LIN {X 0,Y 392.678,Z 1253.285,A -85,B 0,C 180,E1 10734.702,E2 10734.702} C_VEL
LIN {X 0,Y 397.853,Z 1224.84,A -85,B 0,C 180,E1 10739.855,E2 10739.855} C_VEL
LIN {X 0,Y 404.262,Z 1192.64,A -85,B 0,C 180,E1 10744.206,E2 10744.206} C_VEL
LIN {X 0,Y 411.173,Z 1158.01,A -85,B 0,C 180,E1 10747.665,E2 10747.665} C_VEL
LIN {X 0,Y 417.671,Z 1121.351,A -85,B 0,C 180,E1 10750.31,E2 10750.31} C_VEL
LIN {X 0,Y 423.279,Z 1083.5,A -85,B 0,C 180,E1 10752.143,E2 10752.143} C_VEL
LIN {X 0,Y 425.073,Z 1063.403,A -85,B 0,C 180,E1 10752.868,E2 10752.868} C_VEL
LIN {X 0,Y 408.001,Z 1028.181,A -85,B 0,C 180,E1 10756.188,E2 10756.188} C_VEL
LIN {X 0,Y 387.571,Z 994.661,A -85,B 0,C 180,E1 10760.209,E2 10760.209} C_VEL
LIN {X 0,Y 385.179,Z 989.03,A -85,B 0,C 180,E1 10760.945,E2 10760.945} C_VEL
LIN {X 0,Y 385.144,Z 989.03,A -85,B 0,C 180,E1 10766.736,E2 10766.736} C_VEL
LIN {X 0,Y 385.369,Z 989.03,A -85,B 0,C 180,E1 10774.238,E2 10774.238} C_VEL
LIN {X 0,Y 385.666,Z 989.03,A -85,B 0,C 180,E1 10779.892,E2 10779.892} C_VEL
LIN {X 0,Y 385.82,Z 989.03,A -85,B 0,C 180,E1 10786.428,E2 10786.428} C_VEL
LIN {X 0,Y 386.249,Z 989.03,A -85,B 0,C 180,E1 10793.269,E2 10793.269} C_VEL
LIN {X 0,Y 386.525,Z 989.03,A -85,B 0,C 180,E1 10800,E2 10800} C_VEL
LIN {X 0,Y 386.241,Z 989.03,A -85,B 0,C 180,E1 10806.731,E2 10806.731} C_VEL
LIN {X 0,Y 385.972,Z 989.03,A -85,B 0,C 180,E1 10813.566,E2 10813.566} C_VEL
LIN {X 0,Y 385.612,Z 989.03,A -85,B 0,C 180,E1 10820.621,E2 10820.621} C_VEL
LIN {X 0,Y 385.312,Z 989.03,A -85,B 0,C 180,E1 10828.03,E2 10828.03} C_VEL
LIN {X 0,Y 385.061,Z 989.03,A -85,B 0,C 180,E1 10834.619,E2 10834.619} C_VEL
LIN {X 0,Y 385.053,Z 989.03,A -85,B 0,C 180,E1 10838.83,E2 10838.83} C_VEL
LIN {X 0,Y 385.09,Z 989.144,A -85,B 0,C 180,E1 10842.934,E2 10842.934} C_VEL
LIN {X 0,Y 392.046,Z 1004.005,A -85,B 0,C 180,E1 10845.356,E2 10845.356} C_VEL
LIN {X 0,Y 402.939,Z 1029.34,A -85,B 0,C 180,E1 10849.545,E2 10849.545} C_VEL
LIN {X 0,Y 410.17,Z 1055.044,A -85,B 0,C 180,E1 10853.66,E2 10853.66} C_VEL
LIN {X 0,Y 411.018,Z 1064.8,A -85,B 0,C 180,E1 10855.123,E2 10855.123} C_VEL
LIN {X 0,Y 404.003,Z 1094.796,A -85,B 0,C 180,E1 10859.209,E2 10859.209} C_VEL
LIN {X 0,Y 397.397,Z 1120.838,A -85,B 0,C 180,E1 10864.108,E2 10864.108} C_VEL
LIN {X 0,Y 392.663,Z 1140.325,A -85,B 0,C 180,E1 10869.178,E2 10869.178} C_VEL
LIN {X 0,Y 389.485,Z 1155.427,A -85,B 0,C 180,E1 10874.758,E2 10874.758} C_VEL
LIN {X 0,Y 388.053,Z 1164.693,A -85,B 0,C 180,E1 10879.923,E2 10879.923} C_VEL
LIN {X 0,Y 387.281,Z 1170.266,A -85,B 0,C 180,E1 10885.531,E2 10885.531} C_VEL
LIN {X 0,Y 387.373,Z 1171.602,A -85,B 0,C 180,E1 10890.001,E2 10890.001} C_VEL
LIN {X 0,Y 387.286,Z 1170.199,A -85,B 0,C 180,E1 10894.47,E2 10894.47} C_VEL
LIN {X 0,Y 388.016,Z 1164.559,A -85,B 0,C 180,E1 10900.08,E2 10900.08} C_VEL
LIN {X 0,Y 389.699,Z 1154.162,A -85,B 0,C 180,E1 10905.728,E2 10905.728} C_VEL
LIN {X 0,Y 393.119,Z 1138.154,A -85,B 0,C 180,E1 10911.388,E2 10911.388} C_VEL
LIN {X 0,Y 398.156,Z 1117.854,A -85,B 0,C 180,E1 10916.445,E2 10916.445} C_VEL
LIN {X 0,Y 404.626,Z 1091.985,A -85,B 0,C 180,E1 10921.132,E2 10921.132} C_VEL
LIN {X 0,Y 411.178,Z 1062.825,A -85,B 0,C 180,E1 10925.038,E2 10925.038} C_VEL
LIN {X 0,Y 407.077,Z 1042.475,A -85,B 0,C 180,E1 10928.252,E2 10928.252} C_VEL
LIN {X 0,Y 397.567,Z 1015.888,A -85,B 0,C 180,E1 10932.556,E2 10932.556} C_VEL
LIN {X 0,Y 385.142,Z 989.03,A -85,B 0,C 180,E1 10936.979,E2 10936.979} C_VEL
LIN {X 0,Y 385.177,Z 989.03,A -85,B 0,C 180,E1 10944.011,E2 10944.011} C_VEL
LIN {X 0,Y 385.338,Z 989.03,A -85,B 0,C 180,E1 10951.972,E2 10951.972} C_VEL
LIN {X 0,Y 385.624,Z 989.03,A -85,B 0,C 180,E1 10959.38,E2 10959.38} C_VEL
LIN {X 0,Y 385.831,Z 989.03,A -85,B 0,C 180,E1 10966.429,E2 10966.429} C_VEL
LIN {X 0,Y 386.309,Z 989.03,A -85,B 0,C 180,E1 10973.271,E2 10973.271} C_VEL
LIN {X 0,Y 386.585,Z 989.03,A -85,B 0,C 180,E1 10980,E2 10980} C_VEL
LIN {X 0,Y 386.252,Z 989.03,A -85,B 0,C 180,E1 10986.731,E2 10986.731} C_VEL
LIN {X 0,Y 385.983,Z 989.03,A -85,B 0,C 180,E1 10993.566,E2 10993.566} C_VEL
LIN {X 0,Y 385.608,Z 989.03,A -85,B 0,C 180,E1 11000.621,E2 11000.621} C_VEL
LIN {X 0,Y 385.384,Z 989.03,A -85,B 0,C 180,E1 11008.025,E2 11008.025} C_VEL
LIN {X 0,Y 385.21,Z 989.03,A -85,B 0,C 180,E1 11014.648,E2 11014.648} C_VEL
LIN {X 0,Y 385.194,Z 989.03,A -85,B 0,C 180,E1 11019.234,E2 11019.234} C_VEL
LIN {X 0,Y 387.509,Z 994.603,A -85,B 0,C 180,E1 11019.796,E2 11019.796} C_VEL
LIN {X 0,Y 408.246,Z 1028.761,A -85,B 0,C 180,E1 11023.871,E2 11023.871} C_VEL
LIN {X 0,Y 425.015,Z 1063.2,A -85,B 0,C 180,E1 11027.121,E2 11027.121} C_VEL
LIN {X 0,Y 420.317,Z 1104.533,A -85,B 0,C 180,E1 11028.776,E2 11028.776} C_VEL
LIN {X 0,Y 414.189,Z 1141.892,A -85,B 0,C 180,E1 11031.062,E2 11031.062} C_VEL
LIN {X 0,Y 407.588,Z 1176.514,A -85,B 0,C 180,E1 11034.053,E2 11034.053} C_VEL
LIN {X 0,Y 400.807,Z 1210.155,A -85,B 0,C 180,E1 11038.008,E2 11038.008} C_VEL
LIN {X 0,Y 395.066,Z 1240.02,A -85,B 0,C 180,E1 11042.718,E2 11042.718} C_VEL
LIN {X 0,Y 390.9,Z 1264.641,A -85,B 0,C 180,E1 11047.887,E2 11047.887} C_VEL
LIN {X 0,Y 388.53,Z 1283,A -85,B 0,C 180,E1 11053.064,E2 11053.064} C_VEL
LIN {X 0,Y 387.502,Z 1297.201,A -85,B 0,C 180,E1 11058.771,E2 11058.771} C_VEL
LIN {X 0,Y 387.197,Z 1304.359,A -85,B 0,C 180,E1 11063.366,E2 11063.366} C_VEL
LIN {X 0,Y 385.864,Z 1305.49,A -85,B 0,C 180,E1 11064.634,E2 11064.634} C_VEL
LIN {X 0,Y 379.328,Z 1306.601,A -85,B 0,C 180,E1 11068.462,E2 11068.462} C_VEL
LIN {X 0,Y 379.401,Z 1306.453,A -85,B 0,C 180,E1 11072.279,E2 11072.279} C_VEL
LIN {X 0,Y 379.39,Z 1301.51,A -85,B 0,C 180,E1 11078.001,E2 11078.001} C_VEL
LIN {X 0,Y 379.998,Z 1290.877,A -85,B 0,C 180,E1 11083.783,E2 11083.783} C_VEL
LIN {X 0,Y 381.69,Z 1274.153,A -85,B 0,C 180,E1 11089.635,E2 11089.635} C_VEL
LIN {X 0,Y 385.422,Z 1250.417,A -85,B 0,C 180,E1 11095.509,E2 11095.509} C_VEL
LIN {X 0,Y 390.649,Z 1223.372,A -85,B 0,C 180,E1 11100.463,E2 11100.463} C_VEL
LIN {X 0,Y 397.402,Z 1191.356,A -85,B 0,C 180,E1 11104.857,E2 11104.857} C_VEL
LIN {X 0,Y 404.812,Z 1155.988,A -85,B 0,C 180,E1 11108.425,E2 11108.425} C_VEL
LIN {X 0,Y 411.507,Z 1119.923,A -85,B 0,C 180,E1 11111.042,E2 11111.042} C_VEL
LIN {X 0,Y 417.429,Z 1081.556,A -85,B 0,C 180,E1 11112.902,E2 11112.902} C_VEL
LIN {X 0,Y 418.782,Z 1066.088,A -85,B 0,C 180,E1 11113.49,E2 11113.49} C_VEL
LIN {X 0,Y 402.032,Z 1031.104,A -85,B 0,C 180,E1 11116.956,E2 11116.956} C_VEL
LIN {X 0,Y 383.336,Z 1000.326,A -85,B 0,C 180,E1 11120.782,E2 11120.782} C_VEL
LIN {X 0,Y 377.323,Z 990.264,A -85,B 0,C 180,E1 11122.162,E2 11122.162} C_VEL
LIN {X 0,Y 377.229,Z 989.03,A -85,B 0,C 180,E1 11122.226,E2 11122.226} C_VEL
LIN {X 0,Y 377.233,Z 989.03,A -85,B 0,C 180,E1 11128.667,E2 11128.667} C_VEL
LIN {X 0,Y 377.43,Z 989.03,A -85,B 0,C 180,E1 11133.91,E2 11133.91} C_VEL
LIN {X 0,Y 377.64,Z 989.03,A -85,B 0,C 180,E1 11138.923,E2 11138.923} C_VEL
LIN {X 0,Y 377.874,Z 989.03,A -85,B 0,C 180,E1 11146.137,E2 11146.137} C_VEL
LIN {X 0,Y 378.323,Z 989.03,A -85,B 0,C 180,E1 11153.128,E2 11153.128} C_VEL
LIN {X 0,Y 378.624,Z 989.03,A -85,B 0,C 180,E1 11160,E2 11160} C_VEL
LIN {X 0,Y 378.322,Z 989.03,A -85,B 0,C 180,E1 11166.872,E2 11166.872} C_VEL
LIN {X 0,Y 378.018,Z 989.03,A -85,B 0,C 180,E1 11173.857,E2 11173.857} C_VEL
LIN {X 0,Y 377.643,Z 989.03,A -85,B 0,C 180,E1 11181.076,E2 11181.076} C_VEL
LIN {X 0,Y 377.343,Z 989.03,A -85,B 0,C 180,E1 11188.676,E2 11188.676} C_VEL
LIN {X 0,Y 377.155,Z 989.03,A -85,B 0,C 180,E1 11194.064,E2 11194.064} C_VEL
LIN {X 0,Y 377.095,Z 989.479,A -85,B 0,C 180,E1 11201.467,E2 11201.467} C_VEL
LIN {X 0,Y 391.31,Z 1019.042,A -85,B 0,C 180,E1 11206.653,E2 11206.653} C_VEL
LIN {X 0,Y 400.323,Z 1044.65,A -85,B 0,C 180,E1 11210.963,E2 11210.963} C_VEL
LIN {X 0,Y 404.616,Z 1066.185,A -85,B 0,C 180,E1 11214.49,E2 11214.49} C_VEL
LIN {X 0,Y 397.271,Z 1096.179,A -85,B 0,C 180,E1 11218.629,E2 11218.629} C_VEL
LIN {X 0,Y 390.355,Z 1122.22,A -85,B 0,C 180,E1 11223.606,E2 11223.606} C_VEL
LIN {X 0,Y 385.324,Z 1141.71,A -85,B 0,C 180,E1 11228.762,E2 11228.762} C_VEL
LIN {X 0,Y 381.79,Z 1157.451,A -85,B 0,C 180,E1 11234.758,E2 11234.758} C_VEL
LIN {X 0,Y 380.134,Z 1167.499,A -85,B 0,C 180,E1 11240.864,E2 11240.864} C_VEL
LIN {X 0,Y 379.522,Z 1171.638,A -85,B 0,C 180,E1 11245.44,E2 11245.44} C_VEL
LIN {X 0,Y 379.614,Z 1172.971,A -85,B 0,C 180,E1 11250.001,E2 11250.001} C_VEL
LIN {X 0,Y 379.676,Z 1170.163,A -85,B 0,C 180,E1 11256.5,E2 11256.5} C_VEL
LIN {X 0,Y 380.849,Z 1162.362,A -85,B 0,C 180,E1 11262.588,E2 11262.588} C_VEL
LIN {X 0,Y 383.434,Z 1149.827,A -85,B 0,C 180,E1 11268.352,E2 11268.352} C_VEL
LIN {X 0,Y 387.757,Z 1131.796,A -85,B 0,C 180,E1 11273.976,E2 11273.976} C_VEL
LIN {X 0,Y 393.732,Z 1109.441,A -85,B 0,C 180,E1 11278.938,E2 11278.938} C_VEL
LIN {X 0,Y 400.35,Z 1083.862,A -85,B 0,C 180,E1 11283.131,E2 11283.131} C_VEL
LIN {X 0,Y 404.336,Z 1064.316,A -85,B 0,C 180,E1 11285.72,E2 11285.72} C_VEL
LIN {X 0,Y 400.071,Z 1043.899,A -85,B 0,C 180,E1 11289.068,E2 11289.068} C_VEL
LIN {X 0,Y 391.003,Z 1018.6,A -85,B 0,C 180,E1 11293.338,E2 11293.338} C_VEL
LIN {X 0,Y 379.685,Z 994.786,A -85,B 0,C 180,E1 11297.498,E2 11297.498} C_VEL
LIN {X 0,Y 377.155,Z 989.03,A -85,B 0,C 180,E1 11298.525,E2 11298.525} C_VEL
LIN {X 0,Y 377.216,Z 989.03,A -85,B 0,C 180,E1 11305.942,E2 11305.942} C_VEL
LIN {X 0,Y 377.434,Z 989.03,A -85,B 0,C 180,E1 11313.911,E2 11313.911} C_VEL
LIN {X 0,Y 377.655,Z 989.03,A -85,B 0,C 180,E1 11318.924,E2 11318.924} C_VEL
LIN {X 0,Y 377.885,Z 989.03,A -85,B 0,C 180,E1 11326.138,E2 11326.138} C_VEL
LIN {X 0,Y 378.405,Z 989.03,A -85,B 0,C 180,E1 11333.129,E2 11333.129} C_VEL
LIN {X 0,Y 378.683,Z 989.03,A -85,B 0,C 180,E1 11340,E2 11340} C_VEL
LIN {X 0,Y 378.333,Z 989.03,A -85,B 0,C 180,E1 11346.872,E2 11346.872} C_VEL
LIN {X 0,Y 378.029,Z 989.03,A -85,B 0,C 180,E1 11353.857,E2 11353.857} C_VEL
LIN {X 0,Y 377.641,Z 989.03,A -85,B 0,C 180,E1 11361.077,E2 11361.077} C_VEL
LIN {X 0,Y 377.403,Z 989.03,A -85,B 0,C 180,E1 11368.672,E2 11368.672} C_VEL
LIN {X 0,Y 377.292,Z 989.03,A -85,B 0,C 180,E1 11374.05,E2 11374.05} C_VEL
LIN {X 0,Y 377.321,Z 989.611,A -85,B 0,C 180,E1 11377.84,E2 11377.84} C_VEL
LIN {X 0,Y 380.057,Z 995.003,A -85,B 0,C 180,E1 11378.501,E2 11378.501} C_VEL
LIN {X 0,Y 400.986,Z 1029.296,A -85,B 0,C 180,E1 11382.849,E2 11382.849} C_VEL
LIN {X 0,Y 418.304,Z 1064.765,A -85,B 0,C 180,E1 11386.401,E2 11386.401} C_VEL
LIN {X 0,Y 418.675,Z 1070.399,A -85,B 0,C 180,E1 11386.691,E2 11386.691} C_VEL
LIN {X 0,Y 412.876,Z 1111.828,A -85,B 0,C 180,E1 11388.486,E2 11388.486} C_VEL
LIN {X 0,Y 405.747,Z 1151.239,A -85,B 0,C 180,E1 11391.174,E2 11391.174} C_VEL
LIN {X 0,Y 398.548,Z 1186.189,A -85,B 0,C 180,E1 11394.55,E2 11394.55} C_VEL
LIN {X 0,Y 391.833,Z 1217.761,A -85,B 0,C 180,E1 11398.673,E2 11398.673} C_VEL
LIN {X 0,Y 386.115,Z 1246.593,A -85,B 0,C 180,E1 11403.709,E2 11403.709} C_VEL
LIN {X 0,Y 382.498,Z 1268.478,A -85,B 0,C 180,E1 11408.783,E2 11408.783} C_VEL
LIN {X 0,Y 380.326,Z 1286.502,A -85,B 0,C 180,E1 11414.465,E2 11414.465} C_VEL
LIN {X 0,Y 379.59,Z 1297.95,A -85,B 0,C 180,E1 11419.694,E2 11419.694} C_VEL
LIN {X 0,Y 379.327,Z 1305.094,A -85,B 0,C 180,E1 11425.436,E2 11425.436} C_VEL
LIN {X 0,Y 379.328,Z 1306.601,A -85,B 0,C 180,E1 11428.462,E2 11428.462} C_VEL
LIN {X 0,Y 376.834,Z 1306.409,A -85,B 0,C 180,E1 11430.409,E2 11430.409} C_VEL
LIN {X 0,Y 371.491,Z 1304.291,A -85,B 0,C 180,E1 11433.674,E2 11433.674} C_VEL
LIN {X 0,Y 371.563,Z 1300.115,A -85,B 0,C 180,E1 11438.171,E2 11438.171} C_VEL
LIN {X 0,Y 372.166,Z 1289.454,A -85,B 0,C 180,E1 11444.079,E2 11444.079} C_VEL
LIN {X 0,Y 373.98,Z 1272.707,A -85,B 0,C 180,E1 11450.057,E2 11450.057} C_VEL
LIN {X 0,Y 377.958,Z 1248.956,A -85,B 0,C 180,E1 11456.051,E2 11456.051} C_VEL
LIN {X 0,Y 383.467,Z 1222.001,A -85,B 0,C 180,E1 11461.079,E2 11461.079} C_VEL
LIN {X 0,Y 390.717,Z 1189.45,A -85,B 0,C 180,E1 11465.606,E2 11465.606} C_VEL
LIN {X 0,Y 398.389,Z 1154.538,A -85,B 0,C 180,E1 11469.162,E2 11469.162} C_VEL
LIN {X 0,Y 405.632,Z 1117.082,A -85,B 0,C 180,E1 11471.884,E2 11471.884} C_VEL
LIN {X 0,Y 411.834,Z 1078.299,A -85,B 0,C 180,E1 11473.731,E2 11473.731} C_VEL
LIN {X 0,Y 412.469,Z 1068.499,A -85,B 0,C 180,E1 11474.151,E2 11474.151} C_VEL
LIN {X 0,Y 395.577,Z 1032.921,A -85,B 0,C 180,E1 11477.86,E2 11477.86} C_VEL
LIN {X 0,Y 375.761,Z 1000.67,A -85,B 0,C 180,E1 11482.146,E2 11482.146} C_VEL
LIN {X 0,Y 369.433,Z 990.747,A -85,B 0,C 180,E1 11483.68,E2 11483.68} C_VEL
LIN {X 0,Y 369.242,Z 989.03,A -85,B 0,C 180,E1 11483.912,E2 11483.912} C_VEL
LIN {X 0,Y 369.339,Z 989.03,A -85,B 0,C 180,E1 11490.642,E2 11490.642} C_VEL
LIN {X 0,Y 369.557,Z 989.03,A -85,B 0,C 180,E1 11495.901,E2 11495.901} C_VEL
LIN {X 0,Y 369.858,Z 989.03,A -85,B 0,C 180,E1 11503.406,E2 11503.406} C_VEL
LIN {X 0,Y 370.156,Z 989.03,A -85,B 0,C 180,E1 11510.615,E2 11510.615} C_VEL
LIN {X 0,Y 370.749,Z 989.03,A -85,B 0,C 180,E1 11517.667,E2 11517.667} C_VEL
LIN {X 0,Y 370.533,Z 989.03,A -85,B 0,C 180,E1 11524.672,E2 11524.672} C_VEL
LIN {X 0,Y 370.164,Z 989.03,A -85,B 0,C 180,E1 11531.938,E2 11531.938} C_VEL
LIN {X 0,Y 369.792,Z 989.03,A -85,B 0,C 180,E1 11539.053,E2 11539.053} C_VEL
LIN {X 0,Y 369.468,Z 989.03,A -85,B 0,C 180,E1 11546.696,E2 11546.696} C_VEL
LIN {X 0,Y 369.264,Z 989.03,A -85,B 0,C 180,E1 11552.088,E2 11552.088} C_VEL
LIN {X 0,Y 369.151,Z 989.607,A -85,B 0,C 180,E1 11559.881,E2 11559.881} C_VEL
LIN {X 0,Y 383.742,Z 1019.162,A -85,B 0,C 180,E1 11565.402,E2 11565.402} C_VEL
LIN {X 0,Y 392.939,Z 1044.415,A -85,B 0,C 180,E1 11569.837,E2 11569.837} C_VEL
LIN {X 0,Y 397.759,Z 1066.931,A -85,B 0,C 180,E1 11573.672,E2 11573.672} C_VEL
LIN {X 0,Y 392.643,Z 1089.914,A -85,B 0,C 180,E1 11576.831,E2 11576.831} C_VEL
LIN {X 0,Y 385.171,Z 1116.991,A -85,B 0,C 180,E1 11581.64,E2 11581.64} C_VEL
LIN {X 0,Y 379.502,Z 1137.276,A -85,B 0,C 180,E1 11586.571,E2 11586.571} C_VEL
LIN {X 0,Y 375.19,Z 1154.392,A -85,B 0,C 180,E1 11592.444,E2 11592.444} C_VEL
LIN {X 0,Y 372.931,Z 1165.744,A -85,B 0,C 180,E1 11598.328,E2 11598.328} C_VEL
LIN {X 0,Y 372.016,Z 1171.296,A -85,B 0,C 180,E1 11603.011,E2 11603.011} C_VEL
LIN {X 0,Y 371.737,Z 1174.024,A -85,B 0,C 180,E1 11607.674,E2 11607.674} C_VEL
LIN {X 0,Y 371.783,Z 1173.978,A -85,B 0,C 180,E1 11612.327,E2 11612.327} C_VEL
LIN {X 0,Y 372.175,Z 1170.147,A -85,B 0,C 180,E1 11618.159,E2 11618.159} C_VEL
LIN {X 0,Y 373.752,Z 1161.175,A -85,B 0,C 180,E1 11624.316,E2 11624.316} C_VEL
LIN {X 0,Y 377.164,Z 1146.373,A -85,B 0,C 180,E1 11630.488,E2 11630.488} C_VEL
LIN {X 0,Y 382.35,Z 1126.983,A -85,B 0,C 180,E1 11636.025,E2 11636.025} C_VEL
LIN {X 0,Y 388.722,Z 1104.338,A -85,B 0,C 180,E1 11640.704,E2 11640.704} C_VEL
LIN {X 0,Y 396.232,Z 1075.974,A -85,B 0,C 180,E1 11645.012,E2 11645.012} C_VEL
LIN {X 0,Y 397.671,Z 1066.442,A -85,B 0,C 180,E1 11646.315,E2 11646.315} C_VEL
LIN {X 0,Y 392.75,Z 1043.961,A -85,B 0,C 180,E1 11650.15,E2 11650.15} C_VEL
LIN {X 0,Y 383.436,Z 1018.721,A -85,B 0,C 180,E1 11654.589,E2 11654.589} C_VEL
LIN {X 0,Y 372.369,Z 995.305,A -85,B 0,C 180,E1 11658.862,E2 11658.862} C_VEL
LIN {X 0,Y 369.241,Z 989.49,A -85,B 0,C 180,E1 11659.997,E2 11659.997} C_VEL
LIN {X 0,Y 369.316,Z 989.03,A -85,B 0,C 180,E1 11667.917,E2 11667.917} C_VEL
LIN {X 0,Y 369.564,Z 989.03,A -85,B 0,C 180,E1 11675.902,E2 11675.902} C_VEL
LIN {X 0,Y 369.79,Z 989.03,A -85,B 0,C 180,E1 11680.947,E2 11680.947} C_VEL
LIN {X 0,Y 370.058,Z 989.03,A -85,B 0,C 180,E1 11688.236,E2 11688.236} C_VEL
LIN {X 0,Y 370.529,Z 989.03,A -85,B 0,C 180,E1 11695.328,E2 11695.328} C_VEL
LIN {X 0,Y 370.803,Z 989.03,A -85,B 0,C 180,E1 11700,E2 11700} C_VEL
LIN {X 0,Y 370.404,Z 989.03,A -85,B 0,C 180,E1 11707.02,E2 11707.02} C_VEL
LIN {X 0,Y 370.103,Z 989.03,A -85,B 0,C 180,E1 11714.16,E2 11714.16} C_VEL
LIN {X 0,Y 369.7,Z 989.03,A -85,B 0,C 180,E1 11721.552,E2 11721.552} C_VEL
LIN {X 0,Y 369.503,Z 989.03,A -85,B 0,C 180,E1 11726.693,E2 11726.693} C_VEL
LIN {X 0,Y 369.393,Z 989.03,A -85,B 0,C 180,E1 11732.076,E2 11732.076} C_VEL
LIN {X 0,Y 369.305,Z 989.063,A -85,B 0,C 180,E1 11736.266,E2 11736.266} C_VEL
LIN {X 0,Y 371.465,Z 994.405,A -85,B 0,C 180,E1 11736.862,E2 11736.862} C_VEL
LIN {X 0,Y 387.416,Z 1018.882,A -85,B 0,C 180,E1 11740.447,E2 11740.447} C_VEL
LIN {X 0,Y 406.277,Z 1054.027,A -85,B 0,C 180,E1 11744.424,E2 11744.424} C_VEL
LIN {X 0,Y 412.809,Z 1069.578,A -85,B 0,C 180,E1 11745.946,E2 11745.946} C_VEL
LIN {X 0,Y 406.584,Z 1111.78,A -85,B 0,C 180,E1 11747.81,E2 11747.81} C_VEL
LIN {X 0,Y 399.395,Z 1149.944,A -85,B 0,C 180,E1 11750.454,E2 11750.454} C_VEL
LIN {X 0,Y 391.848,Z 1184.794,A -85,B 0,C 180,E1 11753.859,E2 11753.859} C_VEL
LIN {X 0,Y 384.669,Z 1216.732,A -85,B 0,C 180,E1 11758.099,E2 11758.099} C_VEL
LIN {X 0,Y 378.659,Z 1245.134,A -85,B 0,C 180,E1 11763.153,E2 11763.153} C_VEL
LIN {X 0,Y 374.925,Z 1266.574,A -85,B 0,C 180,E1 11768.202,E2 11768.202} C_VEL
LIN {X 0,Y 372.537,Z 1285.073,A -85,B 0,C 180,E1 11774.131,E2 11774.131} C_VEL
LIN {X 0,Y 371.787,Z 1296.55,A -85,B 0,C 180,E1 11779.475,E2 11779.475} C_VEL
LIN {X 0,Y 371.531,Z 1303.714,A -85,B 0,C 180,E1 11785.34,E2 11785.34} C_VEL
LIN {X 0,Y 371.663,Z 1305.551,A -85,B 0,C 180,E1 11789.999,E2 11789.999} C_VEL
LIN {X 0,Y 371.491,Z 1304.291,A -85,B 0,C 180,E1 11793.674,E2 11793.674} C_VEL
LIN {X 0,Y 369.021,Z 1302.501,A -85,B 0,C 180,E1 11795.651,E2 11795.651} C_VEL
LIN {X 0,Y 363.759,Z 1297.873,A -85,B 0,C 180,E1 11798.936,E2 11798.936} C_VEL
LIN {X 0,Y 364.354,Z 1288.032,A -85,B 0,C 180,E1 11804.388,E2 11804.388} C_VEL
LIN {X 0,Y 366.313,Z 1271.266,A -85,B 0,C 180,E1 11810.496,E2 11810.496} C_VEL
LIN {X 0,Y 370.477,Z 1247.485,A -85,B 0,C 180,E1 11816.618,E2 11816.618} C_VEL
LIN {X 0,Y 376.595,Z 1219.606,A -85,B 0,C 180,E1 11821.88,E2 11821.88} C_VEL
LIN {X 0,Y 384.178,Z 1187.324,A -85,B 0,C 180,E1 11826.404,E2 11826.404} C_VEL
LIN {X 0,Y 392.117,Z 1152.504,A -85,B 0,C 180,E1 11829.977,E2 11829.977} C_VEL
LIN {X 0,Y 399.645,Z 1115.662,A -85,B 0,C 180,E1 11832.658,E2 11832.658} C_VEL
LIN {X 0,Y 405.998,Z 1077.62,A -85,B 0,C 180,E1 11834.484,E2 11834.484} C_VEL
LIN {X 0,Y 406.064,Z 1070.652,A -85,B 0,C 180,E1 11834.855,E2 11834.855} C_VEL
LIN {X 0,Y 389.564,Z 1035.608,A -85,B 0,C 180,E1 11838.712,E2 11838.712} C_VEL
LIN {X 0,Y 371.672,Z 1006.271,A -85,B 0,C 180,E1 11842.758,E2 11842.758} C_VEL
LIN {X 0,Y 363.743,Z 994.711,A -85,B 0,C 180,E1 11844.733,E2 11844.733} C_VEL
LIN {X 0,Y 361.301,Z 989.03,A -85,B 0,C 180,E1 11845.494,E2 11845.494} C_VEL
LIN {X 0,Y 361.467,Z 989.03,A -85,B 0,C 180,E1 11852.665,E2 11852.665} C_VEL
LIN {X 0,Y 361.712,Z 989.03,A -85,B 0,C 180,E1 11857.948,E2 11857.948} C_VEL
LIN {X 0,Y 361.995,Z 989.03,A -85,B 0,C 180,E1 11865.516,E2 11865.516} C_VEL
LIN {X 0,Y 362.465,Z 989.03,A -85,B 0,C 180,E1 11872.826,E2 11872.826} C_VEL
LIN {X 0,Y 362.845,Z 989.03,A -85,B 0,C 180,E1 11880,E2 11880} C_VEL
LIN {X 0,Y 362.478,Z 989.03,A -85,B 0,C 180,E1 11887.174,E2 11887.174} C_VEL
LIN {X 0,Y 362.132,Z 989.03,A -85,B 0,C 180,E1 11894.478,E2 11894.478} C_VEL
LIN {X 0,Y 361.715,Z 989.03,A -85,B 0,C 180,E1 11902.052,E2 11902.052} C_VEL
LIN {X 0,Y 361.386,Z 989.03,A -85,B 0,C 180,E1 11910.07,E2 11910.07} C_VEL
LIN {X 0,Y 361.161,Z 989.132,A -85,B 0,C 180,E1 11918.126,E2 11918.126} C_VEL
LIN {X 0,Y 363.518,Z 994.656,A -85,B 0,C 180,E1 11919.12,E2 11919.12} C_VEL
LIN {X 0,Y 375.052,Z 1016.793,A -85,B 0,C 180,E1 11923.597,E2 11923.597} C_VEL
LIN {X 0,Y 385.109,Z 1042.693,A -85,B 0,C 180,E1 11928.37,E2 11928.37} C_VEL
LIN {X 0,Y 390.866,Z 1067.353,A -85,B 0,C 180,E1 11932.759,E2 11932.759} C_VEL
LIN {X 0,Y 390.515,Z 1074.69,A -85,B 0,C 180,E1 11933.88,E2 11933.88} C_VEL
LIN {X 0,Y 382.948,Z 1102.471,A -85,B 0,C 180,E1 11938.027,E2 11938.027} C_VEL
LIN {X 0,Y 375.893,Z 1126.471,A -85,B 0,C 180,E1 11942.899,E2 11942.899} C_VEL
LIN {X 0,Y 370.254,Z 1146.245,A -85,B 0,C 180,E1 11948.482,E2 11948.482} C_VEL
LIN {X 0,Y 366.503,Z 1160.945,A -85,B 0,C 180,E1 11954.478,E2 11954.478} C_VEL
LIN {X 0,Y 364.739,Z 1170.251,A -85,B 0,C 180,E1 11960.475,E2 11960.475} C_VEL
LIN {X 0,Y 364.009,Z 1174.384,A -85,B 0,C 180,E1 11965.245,E2 11965.245} C_VEL
LIN {X 0,Y 364.073,Z 1175.714,A -85,B 0,C 180,E1 11970.001,E2 11970.001} C_VEL
LIN {X 0,Y 364.104,Z 1173.573,A -85,B 0,C 180,E1 11975.944,E2 11975.944} C_VEL
LIN {X 0,Y 365.228,Z 1167.001,A -85,B 0,C 180,E1 11981.923,E2 11981.923} C_VEL
LIN {X 0,Y 367.799,Z 1155.55,A -85,B 0,C 180,E1 11987.922,E2 11987.922} C_VEL
LIN {X 0,Y 372.382,Z 1138.357,A -85,B 0,C 180,E1 11993.907,E2 11993.907} C_VEL
LIN {X 0,Y 379.233,Z 1115.189,A -85,B 0,C 180,E1 11999.5,E2 11999.5} C_VEL
LIN {X 0,Y 386.852,Z 1088.602,A -85,B 0,C 180,E1 12004.107,E2 12004.107} C_VEL
LIN {X 0,Y 391.155,Z 1069.979,A -85,B 0,C 180,E1 12006.7,E2 12006.7} C_VEL
LIN {X 0,Y 386.473,Z 1047.664,A -85,B 0,C 180,E1 12010.641,E2 12010.641} C_VEL
LIN {X 0,Y 377.206,Z 1021.674,A -85,B 0,C 180,E1 12015.385,E2 12015.385} C_VEL
LIN {X 0,Y 365.469,Z 998.139,A -85,B 0,C 180,E1 12020.032,E2 12020.032} C_VEL
LIN {X 0,Y 361.325,Z 989.914,A -85,B 0,C 180,E1 12021.659,E2 12021.659} C_VEL
LIN {X 0,Y 361.24,Z 989.03,A -85,B 0,C 180,E1 12022.533,E2 12022.533} C_VEL
LIN {X 0,Y 361.406,Z 989.03,A -85,B 0,C 180,E1 12029.932,E2 12029.932} C_VEL
LIN {X 0,Y 361.725,Z 989.03,A -85,B 0,C 180,E1 12037.949,E2 12037.949} C_VEL
LIN {X 0,Y 362.007,Z 989.03,A -85,B 0,C 180,E1 12045.517,E2 12045.517} C_VEL
LIN {X 0,Y 362.515,Z 989.03,A -85,B 0,C 180,E1 12053.1,E2 12053.1} C_VEL
LIN {X 0,Y 362.9,Z 989.03,A -85,B 0,C 180,E1 12060,E2 12060} C_VEL
LIN {X 0,Y 362.488,Z 989.03,A -85,B 0,C 180,E1 12067.174,E2 12067.174} C_VEL
LIN {X 0,Y 362.141,Z 989.03,A -85,B 0,C 180,E1 12074.478,E2 12074.478} C_VEL
LIN {X 0,Y 361.716,Z 989.03,A -85,B 0,C 180,E1 12082.052,E2 12082.052} C_VEL
LIN {X 0,Y 361.477,Z 989.03,A -85,B 0,C 180,E1 12090.061,E2 12090.061} C_VEL
LIN {X 0,Y 361.354,Z 989.03,A -85,B 0,C 180,E1 12094.59,E2 12094.59} C_VEL
LIN {X 0,Y 363.676,Z 994.613,A -85,B 0,C 180,E1 12095.276,E2 12095.276} C_VEL
LIN {X 0,Y 373.684,Z 1009.116,A -85,B 0,C 180,E1 12097.735,E2 12097.735} C_VEL
LIN {X 0,Y 392.762,Z 1041.766,A -85,B 0,C 180,E1 12102.022,E2 12102.022} C_VEL
LIN {X 0,Y 406.518,Z 1071.77,A -85,B 0,C 180,E1 12105.271,E2 12105.271} C_VEL
LIN {X 0,Y 400.249,Z 1112.266,A -85,B 0,C 180,E1 12107.144,E2 12107.144} C_VEL
LIN {X 0,Y 393.069,Z 1148.714,A -85,B 0,C 180,E1 12109.713,E2 12109.713} C_VEL
LIN {X 0,Y 385.107,Z 1183.73,A -85,B 0,C 180,E1 12113.181,E2 12113.181} C_VEL
LIN {X 0,Y 377.588,Z 1215.535,A -85,B 0,C 180,E1 12117.477,E2 12117.477} C_VEL
LIN {X 0,Y 371.413,Z 1243.182,A -85,B 0,C 180,E1 12122.473,E2 12122.473} C_VEL
LIN {X 0,Y 367.268,Z 1265.116,A -85,B 0,C 180,E1 12127.723,E2 12127.723} C_VEL
LIN {X 0,Y 364.733,Z 1283.64,A -85,B 0,C 180,E1 12133.783,E2 12133.783} C_VEL
LIN {X 0,Y 363.973,Z 1295.147,A -85,B 0,C 180,E1 12139.247,E2 12139.247} C_VEL
LIN {X 0,Y 363.733,Z 1302.333,A -85,B 0,C 180,E1 12145.24,E2 12145.24} C_VEL
LIN {X 0,Y 363.903,Z 1304.182,A -85,B 0,C 180,E1 12149.999,E2 12149.999} C_VEL
LIN {X 0,Y 363.732,Z 1301.853,A -85,B 0,C 180,E1 12155.35,E2 12155.35} C_VEL
LIN {X 0,Y 363.759,Z 1297.873,A -85,B 0,C 180,E1 12158.936,E2 12158.936} C_VEL
LIN {X 0,Y 361.394,Z 1294.548,A -85,B 0,C 180,E1 12160.907,E2 12160.907} C_VEL
LIN {X 0,Y 356.5,Z 1288.446,A -85,B 0,C 180,E1 12163.835,E2 12163.835} C_VEL
LIN {X 0,Y 356.456,Z 1287.728,A -85,B 0,C 180,E1 12164.173,E2 12164.173} C_VEL
LIN {X 0,Y 358.014,Z 1273.656,A -85,B 0,C 180,E1 12169.705,E2 12169.705} C_VEL
LIN {X 0,Y 361.722,Z 1252.394,A -85,B 0,C 180,E1 12175.713,E2 12175.713} C_VEL
LIN {X 0,Y 367.413,Z 1226.874,A -85,B 0,C 180,E1 12181.049,E2 12181.049} C_VEL
LIN {X 0,Y 374.872,Z 1196.364,A -85,B 0,C 180,E1 12185.813,E2 12185.813} C_VEL
LIN {X 0,Y 383.368,Z 1161.982,A -85,B 0,C 180,E1 12189.747,E2 12189.747} C_VEL
LIN {X 0,Y 391.44,Z 1125.729,A -85,B 0,C 180,E1 12192.719,E2 12192.719} C_VEL
LIN {X 0,Y 398.491,Z 1087.85,A -85,B 0,C 180,E1 12194.818,E2 12194.818} C_VEL
LIN {X 0,Y 400.148,Z 1074.235,A -85,B 0,C 180,E1 12195.42,E2 12195.42} C_VEL
LIN {X 0,Y 383.973,Z 1038.928,A -85,B 0,C 180,E1 12199.49,E2 12199.49} C_VEL
LIN {X 0,Y 365.152,Z 1007.847,A -85,B 0,C 180,E1 12204.015,E2 12204.015} C_VEL
LIN {X 0,Y 355.999,Z 994.891,A -85,B 0,C 180,E1 12206.447,E2 12206.447} C_VEL
LIN {X 0,Y 353.445,Z 989.879,A -85,B 0,C 180,E1 12207.226,E2 12207.226} C_VEL
LIN {X 0,Y 353.36,Z 989.03,A -85,B 0,C 180,E1 12207.527,E2 12207.527} C_VEL
LIN {X 0,Y 353.623,Z 989.03,A -85,B 0,C 180,E1 12214.741,E2 12214.741} C_VEL
LIN {X 0,Y 353.968,Z 989.03,A -85,B 0,C 180,E1 12222.638,E2 12222.638} C_VEL
LIN {X 0,Y 354.289,Z 989.03,A -85,B 0,C 180,E1 12230.191,E2 12230.191} C_VEL
LIN {X 0,Y 354.935,Z 989.03,A -85,B 0,C 180,E1 12237.563,E2 12237.563} C_VEL
LIN {X 0,Y 354.701,Z 989.03,A -85,B 0,C 180,E1 12244.881,E2 12244.881} C_VEL
LIN {X 0,Y 354.344,Z 989.03,A -85,B 0,C 180,E1 12252.294,E2 12252.294} C_VEL
LIN {X 0,Y 353.839,Z 989.03,A -85,B 0,C 180,E1 12260.246,E2 12260.246} C_VEL
LIN {X 0,Y 353.503,Z 989.03,A -85,B 0,C 180,E1 12268.004,E2 12268.004} C_VEL
LIN {X 0,Y 353.251,Z 989.03,A -85,B 0,C 180,E1 12275.745,E2 12275.745} C_VEL
LIN {X 0,Y 353.276,Z 989.701,A -85,B 0,C 180,E1 12276.322,E2 12276.322} C_VEL
LIN {X 0,Y 355.56,Z 994.607,A -85,B 0,C 180,E1 12277.292,E2 12277.292} C_VEL
LIN {X 0,Y 367.765,Z 1017.41,A -85,B 0,C 180,E1 12282.25,E2 12282.25} C_VEL
LIN {X 0,Y 377.993,Z 1043.286,A -85,B 0,C 180,E1 12287.261,E2 12287.261} C_VEL
LIN {X 0,Y 383.983,Z 1067.831,A -85,B 0,C 180,E1 12291.808,E2 12291.808} C_VEL
LIN {X 0,Y 384.289,Z 1075.833,A -85,B 0,C 180,E1 12293.162,E2 12293.162} C_VEL
LIN {X 0,Y 376.464,Z 1103.432,A -85,B 0,C 180,E1 12297.322,E2 12297.322} C_VEL
LIN {X 0,Y 369.085,Z 1127.417,A -85,B 0,C 180,E1 12302.24,E2 12302.24} C_VEL
LIN {X 0,Y 363.471,Z 1145.861,A -85,B 0,C 180,E1 12307.417,E2 12307.417} C_VEL
LIN {X 0,Y 359.246,Z 1161.133,A -85,B 0,C 180,E1 12313.53,E2 12313.53} C_VEL
LIN {X 0,Y 357.306,Z 1170.208,A -85,B 0,C 180,E1 12319.045,E2 12319.045} C_VEL
LIN {X 0,Y 356.258,Z 1175.756,A -85,B 0,C 180,E1 12325.141,E2 12325.141} C_VEL
LIN {X 0,Y 356.292,Z 1177.087,A -85,B 0,C 180,E1 12330.001,E2 12330.001} C_VEL
LIN {X 0,Y 356.258,Z 1175.694,A -85,B 0,C 180,E1 12334.86,E2 12334.86} C_VEL
LIN {X 0,Y 357.28,Z 1170.079,A -85,B 0,C 180,E1 12340.957,E2 12340.957} C_VEL
LIN {X 0,Y 359.602,Z 1159.704,A -85,B 0,C 180,E1 12347.083,E2 12347.083} C_VEL
LIN {X 0,Y 364.008,Z 1143.714,A -85,B 0,C 180,E1 12353.194,E2 12353.194} C_VEL
LIN {X 0,Y 370.443,Z 1122.838,A -85,B 0,C 180,E1 12358.739,E2 12358.739} C_VEL
LIN {X 0,Y 378.089,Z 1097.91,A -85,B 0,C 180,E1 12363.519,E2 12363.519} C_VEL
LIN {X 0,Y 384.584,Z 1073.109,A -85,B 0,C 180,E1 12367.162,E2 12367.162} C_VEL
LIN {X 0,Y 380,Z 1050.557,A -85,B 0,C 180,E1 12371.296,E2 12371.296} C_VEL
LIN {X 0,Y 370.876,Z 1024.593,A -85,B 0,C 180,E1 12376.238,E2 12376.238} C_VEL
LIN {X 0,Y 359.671,Z 1001.338,A -85,B 0,C 180,E1 12381.001,E2 12381.001} C_VEL
LIN {X 0,Y 353.396,Z 990.183,A -85,B 0,C 180,E1 12383.487,E2 12383.487} C_VEL
LIN {X 0,Y 353.322,Z 989.03,A -85,B 0,C 180,E1 12383.806,E2 12383.806} C_VEL
LIN {X 0,Y 353.391,Z 989.03,A -85,B 0,C 180,E1 12389.177,E2 12389.177} C_VEL
LIN {X 0,Y 353.624,Z 989.03,A -85,B 0,C 180,E1 12394.741,E2 12394.741} C_VEL
LIN {X 0,Y 353.984,Z 989.03,A -85,B 0,C 180,E1 12402.639,E2 12402.639} C_VEL
LIN {X 0,Y 354.337,Z 989.03,A -85,B 0,C 180,E1 12410.192,E2 12410.192} C_VEL
LIN {X 0,Y 354.949,Z 989.03,A -85,B 0,C 180,E1 12417.564,E2 12417.564} C_VEL
LIN {X 0,Y 354.711,Z 989.03,A -85,B 0,C 180,E1 12424.881,E2 12424.881} C_VEL
LIN {X 0,Y 354.352,Z 989.03,A -85,B 0,C 180,E1 12432.293,E2 12432.293} C_VEL
LIN {X 0,Y 353.833,Z 989.03,A -85,B 0,C 180,E1 12440.238,E2 12440.238} C_VEL
LIN {X 0,Y 353.558,Z 989.03,A -85,B 0,C 180,E1 12448,E2 12448} C_VEL
LIN {X 0,Y 353.463,Z 989.039,A -85,B 0,C 180,E1 12452.782,E2 12452.782} C_VEL
LIN {X 0,Y 355.612,Z 994.42,A -85,B 0,C 180,E1 12453.478,E2 12453.478} C_VEL
LIN {X 0,Y 358.637,Z 998.56,A -85,B 0,C 180,E1 12454.309,E2 12454.309} C_VEL
LIN {X 0,Y 373.473,Z 1020.921,A -85,B 0,C 180,E1 12458.051,E2 12458.051} C_VEL
LIN {X 0,Y 391.096,Z 1053.194,A -85,B 0,C 180,E1 12462.242,E2 12462.242} C_VEL
LIN {X 0,Y 400.305,Z 1075.124,A -85,B 0,C 180,E1 12464.658,E2 12464.658} C_VEL
LIN {X 0,Y 393.785,Z 1113.743,A -85,B 0,C 180,E1 12466.518,E2 12466.518} C_VEL
LIN {X 0,Y 386.175,Z 1150.205,A -85,B 0,C 180,E1 12469.183,E2 12469.183} C_VEL
LIN {X 0,Y 378.305,Z 1183.117,A -85,B 0,C 180,E1 12472.532,E2 12472.532} C_VEL
LIN {X 0,Y 370.429,Z 1214.677,A -85,B 0,C 180,E1 12476.883,E2 12476.883} C_VEL
LIN {X 0,Y 364.084,Z 1241.718,A -85,B 0,C 180,E1 12481.87,E2 12481.87} C_VEL
LIN {X 0,Y 359.294,Z 1265.593,A -85,B 0,C 180,E1 12487.79,E2 12487.79} C_VEL
LIN {X 0,Y 356.917,Z 1282.202,A -85,B 0,C 180,E1 12493.417,E2 12493.417} C_VEL
LIN {X 0,Y 356.145,Z 1293.74,A -85,B 0,C 180,E1 12499.007,E2 12499.007} C_VEL
LIN {X 0,Y 355.943,Z 1300.953,A -85,B 0,C 180,E1 12505.135,E2 12505.135} C_VEL
LIN {X 0,Y 356.121,Z 1302.808,A -85,B 0,C 180,E1 12509.999,E2 12509.999} C_VEL
LIN {X 0,Y 355.945,Z 1300.958,A -85,B 0,C 180,E1 12514.863,E2 12514.863} C_VEL
LIN {X 0,Y 356.088,Z 1293.734,A -85,B 0,C 180,E1 12520.993,E2 12520.993} C_VEL
LIN {X 0,Y 356.456,Z 1287.728,A -85,B 0,C 180,E1 12524.173,E2 12524.173} C_VEL
LIN {X 0,Y 355.45,Z 1284.749,A -85,B 0,C 180,E1 12525.488,E2 12525.488} C_VEL
LIN {X 0,Y 349.955,Z 1275.428,A -85,B 0,C 180,E1 12529.027,E2 12529.027} C_VEL
LIN {X 0,Y 349.982,Z 1274.529,A -85,B 0,C 180,E1 12529.357,E2 12529.357} C_VEL
LIN {X 0,Y 353.697,Z 1253.658,A -85,B 0,C 180,E1 12535.628,E2 12535.628} C_VEL
LIN {X 0,Y 359.822,Z 1227.302,A -85,B 0,C 180,E1 12541.388,E2 12541.388} C_VEL
LIN {X 0,Y 367.736,Z 1196.603,A -85,B 0,C 180,E1 12546.339,E2 12546.339} C_VEL
LIN {X 0,Y 376.473,Z 1163.028,A -85,B 0,C 180,E1 12550.3,E2 12550.3} C_VEL
LIN {X 0,Y 384.877,Z 1127.292,A -85,B 0,C 180,E1 12553.331,E2 12553.331} C_VEL
LIN {X 0,Y 392.335,Z 1089.369,A -85,B 0,C 180,E1 12555.515,E2 12555.515} C_VEL
LIN {X 0,Y 393.876,Z 1076.75,A -85,B 0,C 180,E1 12556.118,E2 12556.118} C_VEL
LIN {X 0,Y 378.73,Z 1043.045,A -85,B 0,C 180,E1 12560.185,E2 12560.185} C_VEL
LIN {X 0,Y 361.186,Z 1013.549,A -85,B 0,C 180,E1 12564.665,E2 12564.665} C_VEL
LIN {X 0,Y 348.372,Z 995.152,A -85,B 0,C 180,E1 12568.288,E2 12568.288} C_VEL
LIN {X 0,Y 345.555,Z 989.941,A -85,B 0,C 180,E1 12569.216,E2 12569.216} C_VEL
LIN {X 0,Y 345.445,Z 989.03,A -85,B 0,C 180,E1 12569.692,E2 12569.692} C_VEL
LIN {X 0,Y 345.77,Z 989.03,A -85,B 0,C 180,E1 12576.874,E2 12576.874} C_VEL
LIN {X 0,Y 346.122,Z 989.03,A -85,B 0,C 180,E1 12584.836,E2 12584.836} C_VEL
LIN {X 0,Y 346.584,Z 989.03,A -85,B 0,C 180,E1 12592.495,E2 12592.495} C_VEL
LIN {X 0,Y 347.068,Z 989.03,A -85,B 0,C 180,E1 12600,E2 12600} C_VEL
LIN {X 0,Y 346.632,Z 989.03,A -85,B 0,C 180,E1 12607.504,E2 12607.504} C_VEL
LIN {X 0,Y 346.228,Z 989.03,A -85,B 0,C 180,E1 12615.159,E2 12615.159} C_VEL
LIN {X 0,Y 345.777,Z 989.03,A -85,B 0,C 180,E1 12623.126,E2 12623.126} C_VEL
LIN {X 0,Y 345.468,Z 989.03,A -85,B 0,C 180,E1 12629.121,E2 12629.121} C_VEL
LIN {X 0,Y 345.399,Z 989.841,A -85,B 0,C 180,E1 12634.3,E2 12634.3} C_VEL
LIN {X 0,Y 348.328,Z 995.198,A -85,B 0,C 180,E1 12635.553,E2 12635.553} C_VEL
LIN {X 0,Y 361.532,Z 1020.309,A -85,B 0,C 180,E1 12641.297,E2 12641.297} C_VEL
LIN {X 0,Y 371.146,Z 1044.937,A -85,B 0,C 180,E1 12646.277,E2 12646.277} C_VEL
LIN {X 0,Y 377.152,Z 1069.322,A -85,B 0,C 180,E1 12650.979,E2 12650.979} C_VEL
LIN {X 0,Y 377.742,Z 1078.377,A -85,B 0,C 180,E1 12652.608,E2 12652.608} C_VEL
LIN {X 0,Y 369.247,Z 1106.788,A -85,B 0,C 180,E1 12657.022,E2 12657.022} C_VEL
LIN {X 0,Y 361.521,Z 1130.689,A -85,B 0,C 180,E1 12662.129,E2 12662.129} C_VEL
LIN {X 0,Y 355.697,Z 1149.011,A -85,B 0,C 180,E1 12667.555,E2 12667.555} C_VEL
LIN {X 0,Y 351.422,Z 1163.709,A -85,B 0,C 180,E1 12673.794,E2 12673.794} C_VEL
LIN {X 0,Y 349.338,Z 1173.007,A -85,B 0,C 180,E1 12680.051,E2 12680.051} C_VEL
LIN {X 0,Y 348.51,Z 1177.128,A -85,B 0,C 180,E1 12685.033,E2 12685.033} C_VEL
LIN {X 0,Y 348.533,Z 1178.456,A -85,B 0,C 180,E1 12690.001,E2 12690.001} C_VEL
LIN {X 0,Y 348.503,Z 1176.918,A -85,B 0,C 180,E1 12695.221,E2 12695.221} C_VEL
LIN {X 0,Y 349.593,Z 1171.462,A -85,B 0,C 180,E1 12701.201,E2 12701.201} C_VEL
LIN {X 0,Y 352.116,Z 1161.089,A -85,B 0,C 180,E1 12707.458,E2 12707.458} C_VEL
LIN {X 0,Y 356.808,Z 1145.1,A -85,B 0,C 180,E1 12713.69,E2 12713.69} C_VEL
LIN {X 0,Y 363.624,Z 1124.057,A -85,B 0,C 180,E1 12719.373,E2 12719.373} C_VEL
LIN {X 0,Y 371.787,Z 1098.725,A -85,B 0,C 180,E1 12724.274,E2 12724.274} C_VEL
LIN {X 0,Y 377.975,Z 1075.657,A -85,B 0,C 180,E1 12727.735,E2 12727.735} C_VEL
LIN {X 0,Y 373.38,Z 1052.879,A -85,B 0,C 180,E1 12732.089,E2 12732.089} C_VEL
LIN {X 0,Y 364.645,Z 1027.522,A -85,B 0,C 180,E1 12737.103,E2 12737.103} C_VEL
LIN {X 0,Y 354.164,Z 1005.705,A -85,B 0,C 180,E1 12741.846,E2 12741.846} C_VEL
LIN {X 0,Y 345.51,Z 990.232,A -85,B 0,C 180,E1 12745.506,E2 12745.506} C_VEL
LIN {X 0,Y 345.433,Z 989.03,A -85,B 0,C 180,E1 12745.796,E2 12745.796} C_VEL
LIN {X 0,Y 345.686,Z 989.03,A -85,B 0,C 180,E1 12754.119,E2 12754.119} C_VEL
LIN {X 0,Y 346.018,Z 989.03,A -85,B 0,C 180,E1 12762.226,E2 12762.226} C_VEL
LIN {X 0,Y 346.405,Z 989.03,A -85,B 0,C 180,E1 12769.966,E2 12769.966} C_VEL
LIN {X 0,Y 347.05,Z 989.03,A -85,B 0,C 180,E1 12777.508,E2 12777.508} C_VEL
LIN {X 0,Y 346.966,Z 989.03,A -85,B 0,C 180,E1 12782.493,E2 12782.493} C_VEL
LIN {X 0,Y 346.476,Z 989.03,A -85,B 0,C 180,E1 12790.032,E2 12790.032} C_VEL
LIN {X 0,Y 346.071,Z 989.03,A -85,B 0,C 180,E1 12797.771,E2 12797.771} C_VEL
LIN {X 0,Y 345.709,Z 989.03,A -85,B 0,C 180,E1 12805.879,E2 12805.879} C_VEL
LIN {X 0,Y 345.559,Z 989.038,A -85,B 0,C 180,E1 12810.79,E2 12810.79} C_VEL
LIN {X 0,Y 347.624,Z 994.383,A -85,B 0,C 180,E1 12811.53,E2 12811.53} C_VEL
LIN {X 0,Y 350.519,Z 997.898,A -85,B 0,C 180,E1 12812.385,E2 12812.385} C_VEL
LIN {X 0,Y 367.214,Z 1023.01,A -85,B 0,C 180,E1 12816.93,E2 12816.93} C_VEL
LIN {X 0,Y 384.303,Z 1054.463,A -85,B 0,C 180,E1 12821.275,E2 12821.275} C_VEL
LIN {X 0,Y 394.048,Z 1078.271,A -85,B 0,C 180,E1 12824.002,E2 12824.002} C_VEL
LIN {X 0,Y 386.484,Z 1119.436,A -85,B 0,C 180,E1 12826.128,E2 12826.128} C_VEL
LIN {X 0,Y 377.582,Z 1158.21,A -85,B 0,C 180,E1 12829.224,E2 12829.224} C_VEL
LIN {X 0,Y 368.835,Z 1192.599,A -85,B 0,C 180,E1 12833.131,E2 12833.131} C_VEL
LIN {X 0,Y 361.023,Z 1222.761,A -85,B 0,C 180,E1 12837.796,E2 12837.796} C_VEL
LIN {X 0,Y 354.671,Z 1249.291,A -85,B 0,C 180,E1 12843.309,E2 12843.309} C_VEL
LIN {X 0,Y 350.638,Z 1270.281,A -85,B 0,C 180,E1 12849.203,E2 12849.203} C_VEL
LIN {X 0,Y 348.755,Z 1285.183,A -85,B 0,C 180,E1 12854.952,E2 12854.952} C_VEL
LIN {X 0,Y 348.176,Z 1295.936,A -85,B 0,C 180,E1 12861.274,E2 12861.274} C_VEL
LIN {X 0,Y 348.26,Z 1300.951,A -85,B 0,C 180,E1 12867.516,E2 12867.516} C_VEL
LIN {X 0,Y 348.287,Z 1300.957,A -85,B 0,C 180,E1 12872.482,E2 12872.482} C_VEL
LIN {X 0,Y 348.119,Z 1295.932,A -85,B 0,C 180,E1 12878.726,E2 12878.726} C_VEL
LIN {X 0,Y 348.761,Z 1285.188,A -85,B 0,C 180,E1 12885.046,E2 12885.046} C_VEL
LIN {X 0,Y 349.982,Z 1274.529,A -85,B 0,C 180,E1 12889.357,E2 12889.357} C_VEL
LIN {X 0,Y 347.288,Z 1267.042,A -85,B 0,C 180,E1 12891.926,E2 12891.926} C_VEL
LIN {X 0,Y 344.938,Z 1258.631,A -85,B 0,C 180,E1 12894.456,E2 12894.456} C_VEL
LIN {X 0,Y 350.81,Z 1233.493,A -85,B 0,C 180,E1 12900.555,E2 12900.555} C_VEL
LIN {X 0,Y 358.476,Z 1204.827,A -85,B 0,C 180,E1 12905.689,E2 12905.689} C_VEL
LIN {X 0,Y 367.319,Z 1172.692,A -85,B 0,C 180,E1 12909.933,E2 12909.933} C_VEL
LIN {X 0,Y 376.016,Z 1138.423,A -85,B 0,C 180,E1 12913.23,E2 12913.23} C_VEL
LIN {X 0,Y 384.426,Z 1100.226,A -85,B 0,C 180,E1 12915.76,E2 12915.76} C_VEL
LIN {X 0,Y 387.663,Z 1079.348,A -85,B 0,C 180,E1 12916.827,E2 12916.827} C_VEL
LIN {X 0,Y 372.912,Z 1045.961,A -85,B 0,C 180,E1 12921.064,E2 12921.064} C_VEL
LIN {X 0,Y 356.753,Z 1018.527,A -85,B 0,C 180,E1 12925.447,E2 12925.447} C_VEL
LIN {X 0,Y 344.401,Z 1000.743,A -85,B 0,C 180,E1 12929.107,E2 12929.107} C_VEL
LIN {X 0,Y 340.778,Z 995.404,A -85,B 0,C 180,E1 12930.304,E2 12930.304} C_VEL
LIN {X 0,Y 337.723,Z 990.485,A -85,B 0,C 180,E1 12931.386,E2 12931.386} C_VEL
LIN {X 0,Y 337.598,Z 989.03,A -85,B 0,C 180,E1 12931.648,E2 12931.648} C_VEL
LIN {X 0,Y 337.925,Z 989.03,A -85,B 0,C 180,E1 12939.07,E2 12939.07} C_VEL
LIN {X 0,Y 338.315,Z 989.03,A -85,B 0,C 180,E1 12947.114,E2 12947.114} C_VEL
LIN {X 0,Y 338.834,Z 989.03,A -85,B 0,C 180,E1 12954.89,E2 12954.89} C_VEL
LIN {X 0,Y 339.165,Z 989.03,A -85,B 0,C 180,E1 12960,E2 12960} C_VEL
LIN {X 0,Y 338.696,Z 989.03,A -85,B 0,C 180,E1 12967.681,E2 12967.681} C_VEL
LIN {X 0,Y 338.281,Z 989.03,A -85,B 0,C 180,E1 12975.524,E2 12975.524} C_VEL
LIN {X 0,Y 337.937,Z 989.03,A -85,B 0,C 180,E1 12980.929,E2 12980.929} C_VEL
LIN {X 0,Y 337.664,Z 989.03,A -85,B 0,C 180,E1 12986.648,E2 12986.648} C_VEL
LIN {X 0,Y 337.512,Z 989.822,A -85,B 0,C 180,E1 12992.032,E2 12992.032} C_VEL
LIN {X 0,Y 340.487,Z 995.258,A -85,B 0,C 180,E1 12993.439,E2 12993.439} C_VEL
LIN {X 0,Y 353.042,Z 1018.271,A -85,B 0,C 180,E1 12999.163,E2 12999.163} C_VEL
LIN {X 0,Y 363.041,Z 1042.537,A -85,B 0,C 180,E1 13004.434,E2 13004.434} C_VEL
LIN {X 0,Y 369.569,Z 1066.314,A -85,B 0,C 180,E1 13009.21,E2 13009.21} C_VEL
LIN {X 0,Y 371.489,Z 1079.889,A -85,B 0,C 180,E1 13011.889,E2 13011.889} C_VEL
LIN {X 0,Y 362.667,Z 1108.321,A -85,B 0,C 180,E1 13016.379,E2 13016.379} C_VEL
LIN {X 0,Y 354.498,Z 1132.426,A -85,B 0,C 180,E1 13021.628,E2 13021.628} C_VEL
LIN {X 0,Y 347.882,Z 1152.169,A -85,B 0,C 180,E1 13027.695,E2 13027.695} C_VEL
LIN {X 0,Y 343.584,Z 1166.288,A -85,B 0,C 180,E1 13034.069,E2 13034.069} C_VEL
LIN {X 0,Y 341.354,Z 1175.736,A -85,B 0,C 180,E1 13041.1,E2 13041.1} C_VEL
LIN {X 0,Y 340.671,Z 1179.51,A -85,B 0,C 180,E1 13047.462,E2 13047.462} C_VEL
LIN {X 0,Y 340.71,Z 1179.467,A -85,B 0,C 180,E1 13052.539,E2 13052.539} C_VEL
LIN {X 0,Y 341.326,Z 1175.655,A -85,B 0,C 180,E1 13058.902,E2 13058.902} C_VEL
LIN {X 0,Y 343.612,Z 1166.108,A -85,B 0,C 180,E1 13065.932,E2 13065.932} C_VEL
LIN {X 0,Y 347.904,Z 1151.911,A -85,B 0,C 180,E1 13072.305,E2 13072.305} C_VEL
LIN {X 0,Y 354.036,Z 1133.676,A -85,B 0,C 180,E1 13077.961,E2 13077.961} C_VEL
LIN {X 0,Y 361.976,Z 1110.378,A -85,B 0,C 180,E1 13083.144,E2 13083.144} C_VEL
LIN {X 0,Y 370.782,Z 1082.629,A -85,B 0,C 180,E1 13087.625,E2 13087.625} C_VEL
LIN {X 0,Y 371.051,Z 1074.907,A -85,B 0,C 180,E1 13088.98,E2 13088.98} C_VEL
LIN {X 0,Y 365.501,Z 1050.386,A -85,B 0,C 180,E1 13093.867,E2 13093.867} C_VEL
LIN {X 0,Y 356.459,Z 1025.634,A -85,B 0,C 180,E1 13099.047,E2 13099.047} C_VEL
LIN {X 0,Y 344.722,Z 1002.196,A -85,B 0,C 180,E1 13104.55,E2 13104.55} C_VEL
LIN {X 0,Y 339.533,Z 994.302,A -85,B 0,C 180,E1 13106.795,E2 13106.795} C_VEL
LIN {X 0,Y 337.537,Z 989.03,A -85,B 0,C 180,E1 13108.151,E2 13108.151} C_VEL
LIN {X 0,Y 337.849,Z 989.03,A -85,B 0,C 180,E1 13116.299,E2 13116.299} C_VEL
LIN {X 0,Y 338.051,Z 989.03,A -85,B 0,C 180,E1 13121.793,E2 13121.793} C_VEL
LIN {X 0,Y 338.462,Z 989.03,A -85,B 0,C 180,E1 13129.728,E2 13129.728} C_VEL
LIN {X 0,Y 339.132,Z 989.03,A -85,B 0,C 180,E1 13137.45,E2 13137.45} C_VEL
LIN {X 0,Y 339.053,Z 989.03,A -85,B 0,C 180,E1 13142.551,E2 13142.551} C_VEL
LIN {X 0,Y 338.538,Z 989.03,A -85,B 0,C 180,E1 13150.27,E2 13150.27} C_VEL
LIN {X 0,Y 338.093,Z 989.03,A -85,B 0,C 180,E1 13158.205,E2 13158.205} C_VEL
LIN {X 0,Y 337.85,Z 989.03,A -85,B 0,C 180,E1 13163.701,E2 13163.701} C_VEL
LIN {X 0,Y 337.693,Z 989.679,A -85,B 0,C 180,E1 13168.618,E2 13168.618} C_VEL
LIN {X 0,Y 340.141,Z 994.82,A -85,B 0,C 180,E1 13169.536,E2 13169.536} C_VEL
LIN {X 0,Y 342.689,Z 997.754,A -85,B 0,C 180,E1 13170.359,E2 13170.359} C_VEL
LIN {X 0,Y 359.233,Z 1022.093,A -85,B 0,C 180,E1 13175.26,E2 13175.26} C_VEL
LIN {X 0,Y 376.738,Z 1053.874,A -85,B 0,C 180,E1 13180.026,E2 13180.026} C_VEL
LIN {X 0,Y 387.899,Z 1080.19,A -85,B 0,C 180,E1 13183.275,E2 13183.275} C_VEL
LIN {X 0,Y 380.17,Z 1120.158,A -85,B 0,C 180,E1 13185.428,E2 13185.428} C_VEL
LIN {X 0,Y 371.473,Z 1156.542,A -85,B 0,C 180,E1 13188.377,E2 13188.377} C_VEL
LIN {X 0,Y 362.3,Z 1190.888,A -85,B 0,C 180,E1 13192.31,E2 13192.31} C_VEL
LIN {X 0,Y 353.968,Z 1221.281,A -85,B 0,C 180,E1 13197.073,E2 13197.073} C_VEL
LIN {X 0,Y 347.382,Z 1247.092,A -85,B 0,C 180,E1 13202.51,E2 13202.51} C_VEL
LIN {X 0,Y 343.196,Z 1267.54,A -85,B 0,C 180,E1 13208.277,E2 13208.277} C_VEL
LIN {X 0,Y 340.939,Z 1283.753,A -85,B 0,C 180,E1 13214.599,E2 13214.599} C_VEL
LIN {X 0,Y 340.35,Z 1294.538,A -85,B 0,C 180,E1 13221.072,E2 13221.072} C_VEL
LIN {X 0,Y 340.46,Z 1299.573,A -85,B 0,C 180,E1 13227.459,E2 13227.459} C_VEL
LIN {X 0,Y 340.504,Z 1299.583,A -85,B 0,C 180,E1 13232.539,E2 13232.539} C_VEL
LIN {X 0,Y 340.292,Z 1294.535,A -85,B 0,C 180,E1 13238.928,E2 13238.928} C_VEL
LIN {X 0,Y 340.959,Z 1283.761,A -85,B 0,C 180,E1 13245.399,E2 13245.399} C_VEL
LIN {X 0,Y 343.202,Z 1267.514,A -85,B 0,C 180,E1 13251.735,E2 13251.735} C_VEL
LIN {X 0,Y 344.938,Z 1258.631,A -85,B 0,C 180,E1 13254.456,E2 13254.456} C_VEL
LIN {X 0,Y 342.971,Z 1249.792,A -85,B 0,C 180,E1 13256.958,E2 13256.958} C_VEL
LIN {X 0,Y 341.502,Z 1240.314,A -85,B 0,C 180,E1 13259.417,E2 13259.417} C_VEL
LIN {X 0,Y 349.184,Z 1212.421,A -85,B 0,C 180,E1 13264.991,E2 13264.991} C_VEL
LIN {X 0,Y 358.176,Z 1181.299,A -85,B 0,C 180,E1 13269.569,E2 13269.569} C_VEL
LIN {X 0,Y 367.513,Z 1146.926,A -85,B 0,C 180,E1 13273.25,E2 13273.25} C_VEL
LIN {X 0,Y 376.398,Z 1110.099,A -85,B 0,C 180,E1 13275.998,E2 13275.998} C_VEL
LIN {X 0,Y 381.486,Z 1082.244,A -85,B 0,C 180,E1 13277.507,E2 13277.507} C_VEL
LIN {X 0,Y 367.36,Z 1049.585,A -85,B 0,C 180,E1 13281.863,E2 13281.863} C_VEL
LIN {X 0,Y 351.149,Z 1021.25,A -85,B 0,C 180,E1 13286.612,E2 13286.612} C_VEL
LIN {X 0,Y 337.458,Z 1001.75,A -85,B 0,C 180,E1 13290.995,E2 13290.995} C_VEL
LIN {X 0,Y 333.249,Z 995.624,A -85,B 0,C 180,E1 13292.53,E2 13292.53} C_VEL
LIN {X 0,Y 329.99,Z 990.92,A -85,B 0,C 180,E1 13293.798,E2 13293.798} C_VEL
LIN {X 0,Y 329.763,Z 989.03,A -85,B 0,C 180,E1 13294.053,E2 13294.053} C_VEL
LIN {X 0,Y 330.086,Z 989.03,A -85,B 0,C 180,E1 13301.337,E2 13301.337} C_VEL
LIN {X 0,Y 330.505,Z 989.03,A -85,B 0,C 180,E1 13309.477,E2 13309.477} C_VEL
LIN {X 0,Y 331.198,Z 989.03,A -85,B 0,C 180,E1 13317.389,E2 13317.389} C_VEL
LIN {X 0,Y 331.131,Z 989.03,A -85,B 0,C 180,E1 13322.612,E2 13322.612} C_VEL
LIN {X 0,Y 330.613,Z 989.03,A -85,B 0,C 180,E1 13330.519,E2 13330.519} C_VEL
LIN {X 0,Y 330.138,Z 989.03,A -85,B 0,C 180,E1 13338.66,E2 13338.66} C_VEL
LIN {X 0,Y 329.833,Z 989.03,A -85,B 0,C 180,E1 13344.314,E2 13344.314} C_VEL
LIN {X 0,Y 329.664,Z 989.506,A -85,B 0,C 180,E1 13349.461,E2 13349.461} C_VEL
LIN {X 0,Y 332.12,Z 994.858,A -85,B 0,C 180,E1 13350.855,E2 13350.855} C_VEL
LIN {X 0,Y 334.296,Z 998.33,A -85,B 0,C 180,E1 13351.905,E2 13351.905} C_VEL
LIN {X 0,Y 343.312,Z 1013.881,A -85,B 0,C 180,E1 13356.26,E2 13356.26} C_VEL
LIN {X 0,Y 353.816,Z 1037.259,A -85,B 0,C 180,E1 13361.787,E2 13361.787} C_VEL
LIN {X 0,Y 361.135,Z 1060.205,A -85,B 0,C 180,E1 13366.71,E2 13366.71} C_VEL
LIN {X 0,Y 364.886,Z 1081.374,A -85,B 0,C 180,E1 13371.071,E2 13371.071} C_VEL
LIN {X 0,Y 356.753,Z 1108.046,A -85,B 0,C 180,E1 13375.375,E2 13375.375} C_VEL
LIN {X 0,Y 348.191,Z 1132.142,A -85,B 0,C 180,E1 13380.581,E2 13380.581} C_VEL
LIN {X 0,Y 341.219,Z 1151.782,A -85,B 0,C 180,E1 13386.547,E2 13386.547} C_VEL
LIN {X 0,Y 336.383,Z 1166.475,A -85,B 0,C 180,E1 13393.048,E2 13393.048} C_VEL
LIN {X 0,Y 333.957,Z 1175.763,A -85,B 0,C 180,E1 13399.588,E2 13399.588} C_VEL
LIN {X 0,Y 332.928,Z 1180.293,A -85,B 0,C 180,E1 13405.647,E2 13405.647} C_VEL
LIN {X 0,Y 332.994,Z 1181.199,A -85,B 0,C 180,E1 13410.001,E2 13410.001} C_VEL
LIN {X 0,Y 333.012,Z 1179.813,A -85,B 0,C 180,E1 13415.201,E2 13415.201} C_VEL
LIN {X 0,Y 334.254,Z 1174.226,A -85,B 0,C 180,E1 13421.722,E2 13421.722} C_VEL
LIN {X 0,Y 337.175,Z 1163.862,A -85,B 0,C 180,E1 13428.258,E2 13428.258} C_VEL
LIN {X 0,Y 342.278,Z 1148.45,A -85,B 0,C 180,E1 13434.562,E2 13434.562} C_VEL
LIN {X 0,Y 349.886,Z 1127.333,A -85,B 0,C 180,E1 13440.513,E2 13440.513} C_VEL
LIN {X 0,Y 358.833,Z 1101.89,A -85,B 0,C 180,E1 13445.615,E2 13445.615} C_VEL
LIN {X 0,Y 364.9,Z 1082.419,A -85,B 0,C 180,E1 13448.625,E2 13448.625} C_VEL
LIN {X 0,Y 360.881,Z 1059.754,A -85,B 0,C 180,E1 13453.305,E2 13453.305} C_VEL
LIN {X 0,Y 353.062,Z 1035.389,A -85,B 0,C 180,E1 13458.513,E2 13458.513} C_VEL
LIN {X 0,Y 342.732,Z 1012.929,A -85,B 0,C 180,E1 13463.882,E2 13463.882} C_VEL
LIN {X 0,Y 332.428,Z 995.101,A -85,B 0,C 180,E1 13468.879,E2 13468.879} C_VEL
LIN {X 0,Y 329.686,Z 989.749,A -85,B 0,C 180,E1 13470.364,E2 13470.364} C_VEL
LIN {X 0,Y 329.936,Z 989.03,A -85,B 0,C 180,E1 13476.17,E2 13476.17} C_VEL
LIN {X 0,Y 330.223,Z 989.03,A -85,B 0,C 180,E1 13484.088,E2 13484.088} C_VEL
LIN {X 0,Y 330.782,Z 989.03,A -85,B 0,C 180,E1 13492.134,E2 13492.134} C_VEL
LIN {X 0,Y 331.37,Z 989.03,A -85,B 0,C 180,E1 13500,E2 13500} C_VEL
LIN {X 0,Y 330.772,Z 989.03,A -85,B 0,C 180,E1 13507.866,E2 13507.866} C_VEL
LIN {X 0,Y 330.315,Z 989.03,A -85,B 0,C 180,E1 13515.908,E2 13515.908} C_VEL
LIN {X 0,Y 329.845,Z 989.03,A -85,B 0,C 180,E1 13524.313,E2 13524.313} C_VEL
LIN {X 0,Y 329.796,Z 989.512,A -85,B 0,C 180,E1 13526.128,E2 13526.128} C_VEL
LIN {X 0,Y 332.293,Z 994.816,A -85,B 0,C 180,E1 13527.184,E2 13527.184} C_VEL
LIN {X 0,Y 334.952,Z 997.76,A -85,B 0,C 180,E1 13528.139,E2 13528.139} C_VEL
LIN {X 0,Y 349.606,Z 1019.138,A -85,B 0,C 180,E1 13532.968,E2 13532.968} C_VEL
LIN {X 0,Y 363.884,Z 1043.025,A -85,B 0,C 180,E1 13537.146,E2 13537.146} C_VEL
LIN {X 0,Y 378.191,Z 1073.865,A -85,B 0,C 180,E1 13541.439,E2 13541.439} C_VEL
LIN {X 0,Y 381.589,Z 1084.005,A -85,B 0,C 180,E1 13542.645,E2 13542.645} C_VEL
LIN {X 0,Y 373.709,Z 1121.671,A -85,B 0,C 180,E1 13544.756,E2 13544.756} C_VEL
LIN {X 0,Y 364.34,Z 1158.858,A -85,B 0,C 180,E1 13547.897,E2 13547.897} C_VEL
LIN {X 0,Y 355.036,Z 1191.923,A -85,B 0,C 180,E1 13551.838,E2 13551.838} C_VEL
LIN {X 0,Y 346.53,Z 1221.523,A -85,B 0,C 180,E1 13556.647,E2 13556.647} C_VEL
LIN {X 0,Y 339.46,Z 1248.008,A -85,B 0,C 180,E1 13562.468,E2 13562.468} C_VEL
LIN {X 0,Y 334.951,Z 1269.301,A -85,B 0,C 180,E1 13568.873,E2 13568.873} C_VEL
LIN {X 0,Y 332.909,Z 1284.927,A -85,B 0,C 180,E1 13575.563,E2 13575.563} C_VEL
LIN {X 0,Y 332.556,Z 1293.145,A -85,B 0,C 180,E1 13580.861,E2 13580.861} C_VEL
LIN {X 0,Y 332.659,Z 1298.195,A -85,B 0,C 180,E1 13587.399,E2 13587.399} C_VEL
LIN {X 0,Y 332.707,Z 1298.205,A -85,B 0,C 180,E1 13592.599,E2 13592.599} C_VEL
LIN {X 0,Y 332.499,Z 1294.547,A -85,B 0,C 180,E1 13597.824,E2 13597.824} C_VEL
LIN {X 0,Y 332.822,Z 1286.214,A -85,B 0,C 180,E1 13603.77,E2 13603.77} C_VEL
LIN {X 0,Y 334.625,Z 1271.216,A -85,B 0,C 180,E1 13610.455,E2 13610.455} C_VEL
LIN {X 0,Y 339.108,Z 1249.596,A -85,B 0,C 180,E1 13617.133,E2 13617.133} C_VEL
LIN {X 0,Y 341.502,Z 1240.314,A -85,B 0,C 180,E1 13619.417,E2 13619.417} C_VEL
LIN {X 0,Y 340.354,Z 1230.331,A -85,B 0,C 180,E1 13621.833,E2 13621.833} C_VEL
LIN {X 0,Y 339.685,Z 1219.766,A -85,B 0,C 180,E1 13624.187,E2 13624.187} C_VEL
LIN {X 0,Y 348.789,Z 1189.704,A -85,B 0,C 180,E1 13629.118,E2 13629.118} C_VEL
LIN {X 0,Y 358.688,Z 1156.056,A -85,B 0,C 180,E1 13633.128,E2 13633.128} C_VEL
LIN {X 0,Y 368.372,Z 1119.231,A -85,B 0,C 180,E1 13636.212,E2 13636.212} C_VEL
LIN {X 0,Y 375.583,Z 1085.971,A -85,B 0,C 180,E1 13638.116,E2 13638.116} C_VEL
LIN {X 0,Y 362.535,Z 1054.634,A -85,B 0,C 180,E1 13642.464,E2 13642.464} C_VEL
LIN {X 0,Y 347.78,Z 1027.724,A -85,B 0,C 180,E1 13647.115,E2 13647.115} C_VEL
LIN {X 0,Y 333.407,Z 1006.773,A -85,B 0,C 180,E1 13651.995,E2 13651.995} C_VEL
LIN {X 0,Y 329.102,Z 1000.992,A -85,B 0,C 180,E1 13653.629,E2 13653.629} C_VEL
LIN {X 0,Y 326.023,Z 995.985,A -85,B 0,C 180,E1 13654.926,E2 13654.926} C_VEL
LIN {X 0,Y 322.276,Z 991.149,A -85,B 0,C 180,E1 13656.56,E2 13656.56} C_VEL
LIN {X 0,Y 321.991,Z 989.03,A -85,B 0,C 180,E1 13656.828,E2 13656.828} C_VEL
LIN {X 0,Y 322.263,Z 989.03,A -85,B 0,C 180,E1 13663.684,E2 13663.684} C_VEL
LIN {X 0,Y 322.764,Z 989.03,A -85,B 0,C 180,E1 13671.937,E2 13671.937} C_VEL
LIN {X 0,Y 323.278,Z 989.03,A -85,B 0,C 180,E1 13677.325,E2 13677.325} C_VEL
LIN {X 0,Y 323.215,Z 989.03,A -85,B 0,C 180,E1 13682.676,E2 13682.676} C_VEL
LIN {X 0,Y 322.658,Z 989.03,A -85,B 0,C 180,E1 13690.853,E2 13690.853} C_VEL
LIN {X 0,Y 322.351,Z 989.03,A -85,B 0,C 180,E1 13696.312,E2 13696.312} C_VEL
LIN {X 0,Y 322.014,Z 989.03,A -85,B 0,C 180,E1 13702.017,E2 13702.017} C_VEL
LIN {X 0,Y 321.759,Z 989.456,A -85,B 0,C 180,E1 13706.556,E2 13706.556} C_VEL
LIN {X 0,Y 324.336,Z 994.89,A -85,B 0,C 180,E1 13708.147,E2 13708.147} C_VEL
LIN {X 0,Y 326.469,Z 997.976,A -85,B 0,C 180,E1 13709.282,E2 13709.282} C_VEL
LIN {X 0,Y 334.221,Z 1011.231,A -85,B 0,C 180,E1 13713.368,E2 13713.368} C_VEL
LIN {X 0,Y 344.437,Z 1032.022,A -85,B 0,C 180,E1 13718.88,E2 13718.88} C_VEL
LIN {X 0,Y 352.482,Z 1054.702,A -85,B 0,C 180,E1 13724.121,E2 13724.121} C_VEL
LIN {X 0,Y 357.704,Z 1078.354,A -85,B 0,C 180,E1 13729.226,E2 13729.226} C_VEL
LIN {X 0,Y 357.855,Z 1087.687,A -85,B 0,C 180,E1 13731.068,E2 13731.068} C_VEL
LIN {X 0,Y 347.74,Z 1116.575,A -85,B 0,C 180,E1 13736.034,E2 13736.034} C_VEL
LIN {X 0,Y 339.281,Z 1139.09,A -85,B 0,C 180,E1 13741.438,E2 13741.438} C_VEL
LIN {X 0,Y 332.766,Z 1156.635,A -85,B 0,C 180,E1 13747.329,E2 13747.329} C_VEL
LIN {X 0,Y 328.176,Z 1170.156,A -85,B 0,C 180,E1 13753.986,E2 13753.986} C_VEL
LIN {X 0,Y 325.941,Z 1178.49,A -85,B 0,C 180,E1 13760.676,E2 13760.676} C_VEL
LIN {X 0,Y 325.129,Z 1182.255,A -85,B 0,C 180,E1 13767.341,E2 13767.341} C_VEL
LIN {X 0,Y 325.184,Z 1182.21,A -85,B 0,C 180,E1 13772.661,E2 13772.661} C_VEL
LIN {X 0,Y 325.916,Z 1178.41,A -85,B 0,C 180,E1 13779.327,E2 13779.327} C_VEL
LIN {X 0,Y 328.571,Z 1168.876,A -85,B 0,C 180,E1 13786.682,E2 13786.682} C_VEL
LIN {X 0,Y 333.404,Z 1154.69,A -85,B 0,C 180,E1 13793.331,E2 13793.331} C_VEL
LIN {X 0,Y 340.779,Z 1135.108,A -85,B 0,C 180,E1 13799.547,E2 13799.547} C_VEL
LIN {X 0,Y 349.708,Z 1111.109,A -85,B 0,C 180,E1 13804.933,E2 13804.933} C_VEL
LIN {X 0,Y 358.4,Z 1085.425,A -85,B 0,C 180,E1 13809.167,E2 13809.167} C_VEL
LIN {X 0,Y 354.49,Z 1062.418,A -85,B 0,C 180,E1 13814.096,E2 13814.096} C_VEL
LIN {X 0,Y 347.265,Z 1038.962,A -85,B 0,C 180,E1 13819.324,E2 13819.324} C_VEL
LIN {X 0,Y 337.951,Z 1018.256,A -85,B 0,C 180,E1 13824.518,E2 13824.518} C_VEL
LIN {X 0,Y 329.627,Z 1002.421,A -85,B 0,C 180,E1 13829.003,E2 13829.003} C_VEL
LIN {X 0,Y 326.057,Z 996.492,A -85,B 0,C 180,E1 13830.886,E2 13830.886} C_VEL
LIN {X 0,Y 322.003,Z 990.838,A -85,B 0,C 180,E1 13833.048,E2 13833.048} C_VEL
LIN {X 0,Y 321.763,Z 989.03,A -85,B 0,C 180,E1 13833.509,E2 13833.509} C_VEL
LIN {X 0,Y 322.124,Z 989.03,A -85,B 0,C 180,E1 13840.858,E2 13840.858} C_VEL
LIN {X 0,Y 322.595,Z 989.03,A -85,B 0,C 180,E1 13849.216,E2 13849.216} C_VEL
LIN {X 0,Y 323.293,Z 989.03,A -85,B 0,C 180,E1 13857.325,E2 13857.325} C_VEL
LIN {X 0,Y 323.232,Z 989.03,A -85,B 0,C 180,E1 13862.676,E2 13862.676} C_VEL
LIN {X 0,Y 322.666,Z 989.03,A -85,B 0,C 180,E1 13870.85,E2 13870.85} C_VEL
LIN {X 0,Y 322.357,Z 989.03,A -85,B 0,C 180,E1 13876.311,E2 13876.311} C_VEL
LIN {X 0,Y 322.024,Z 989.3,A -85,B 0,C 180,E1 13883.315,E2 13883.315} C_VEL
LIN {X 0,Y 324.127,Z 994.456,A -85,B 0,C 180,E1 13884.375,E2 13884.375} C_VEL
LIN {X 0,Y 327.356,Z 997.951,A -85,B 0,C 180,E1 13885.695,E2 13885.695} C_VEL
LIN {X 0,Y 340.841,Z 1017.002,A -85,B 0,C 180,E1 13890.66,E2 13890.66} C_VEL
LIN {X 0,Y 356.703,Z 1043.147,A -85,B 0,C 180,E1 13895.718,E2 13895.718} C_VEL
LIN {X 0,Y 370.876,Z 1073.497,A -85,B 0,C 180,E1 13900.248,E2 13900.248} C_VEL
LIN {X 0,Y 375.423,Z 1086.703,A -85,B 0,C 180,E1 13901.927,E2 13901.927} C_VEL
LIN {X 0,Y 366.235,Z 1127.826,A -85,B 0,C 180,E1 13904.405,E2 13904.405} C_VEL
LIN {X 0,Y 356.284,Z 1164.539,A -85,B 0,C 180,E1 13907.767,E2 13907.767} C_VEL
LIN {X 0,Y 346.262,Z 1197.935,A -85,B 0,C 180,E1 13912.088,E2 13912.088} C_VEL
LIN {X 0,Y 337.671,Z 1226.672,A -85,B 0,C 180,E1 13917.189,E2 13917.189} C_VEL
LIN {X 0,Y 330.815,Z 1251.769,A -85,B 0,C 180,E1 13923.226,E2 13923.226} C_VEL
LIN {X 0,Y 326.689,Z 1271.484,A -85,B 0,C 180,E1 13929.73,E2 13929.73} C_VEL
LIN {X 0,Y 324.933,Z 1285.899,A -85,B 0,C 180,E1 13936.572,E2 13936.572} C_VEL
LIN {X 0,Y 324.716,Z 1293.153,A -85,B 0,C 180,E1 13941.985,E2 13941.985} C_VEL
LIN {X 0,Y 324.886,Z 1296.821,A -85,B 0,C 180,E1 13947.337,E2 13947.337} C_VEL
LIN {X 0,Y 324.928,Z 1296.831,A -85,B 0,C 180,E1 13952.661,E2 13952.661} C_VEL
LIN {X 0,Y 324.67,Z 1293.153,A -85,B 0,C 180,E1 13958.014,E2 13958.014} C_VEL
LIN {X 0,Y 325.011,Z 1284.794,A -85,B 0,C 180,E1 13964.107,E2 13964.107} C_VEL
LIN {X 0,Y 326.952,Z 1269.77,A -85,B 0,C 180,E1 13970.958,E2 13970.958} C_VEL
LIN {X 0,Y 331.692,Z 1248.123,A -85,B 0,C 180,E1 13977.791,E2 13977.791} C_VEL
LIN {X 0,Y 339.082,Z 1221.802,A -85,B 0,C 180,E1 13983.798,E2 13983.798} C_VEL
LIN {X 0,Y 339.685,Z 1219.766,A -85,B 0,C 180,E1 13984.187,E2 13984.187} C_VEL
LIN {X 0,Y 339.429,Z 1208.671,A -85,B 0,C 180,E1 13986.481,E2 13986.481} C_VEL
LIN {X 0,Y 339.139,Z 1198.597,A -85,B 0,C 180,E1 13988.442,E2 13988.442} C_VEL
LIN {X 0,Y 339.578,Z 1197.029,A -85,B 0,C 180,E1 13988.693,E2 13988.693} C_VEL
LIN {X 0,Y 349.875,Z 1164.414,A -85,B 0,C 180,E1 13992.993,E2 13992.993} C_VEL
LIN {X 0,Y 360.057,Z 1128.756,A -85,B 0,C 180,E1 13996.33,E2 13996.33} C_VEL
LIN {X 0,Y 368.954,Z 1091.595,A -85,B 0,C 180,E1 13998.678,E2 13998.678} C_VEL
LIN {X 0,Y 368.743,Z 1087.001,A -85,B 0,C 180,E1 13999.1,E2 13999.1} C_VEL
LIN {X 0,Y 356.567,Z 1057.224,A -85,B 0,C 180,E1 14003.454,E2 14003.454} C_VEL
LIN {X 0,Y 342.965,Z 1032.306,A -85,B 0,C 180,E1 14008.024,E2 14008.024} C_VEL
LIN {X 0,Y 328.239,Z 1009.736,A -85,B 0,C 180,E1 14013.476,E2 14013.476} C_VEL
LIN {X 0,Y 322.64,Z 1002.35,A -85,B 0,C 180,E1 14015.844,E2 14015.844} C_VEL
LIN {X 0,Y 318.259,Z 995.986,A -85,B 0,C 180,E1 14017.914,E2 14017.914} C_VEL
LIN {X 0,Y 314.428,Z 991.184,A -85,B 0,C 180,E1 14019.885,E2 14019.885} C_VEL
LIN {X 0,Y 314.151,Z 989.03,A -85,B 0,C 180,E1 14020.353,E2 14020.353} C_VEL
LIN {X 0,Y 314.452,Z 989.03,A -85,B 0,C 180,E1 14026.117,E2 14026.117} C_VEL
LIN {X 0,Y 315.063,Z 989.03,A -85,B 0,C 180,E1 14034.503,E2 14034.503} C_VEL
LIN {X 0,Y 315.477,Z 989.03,A -85,B 0,C 180,E1 14040,E2 14040} C_VEL
LIN {X 0,Y 314.906,Z 989.03,A -85,B 0,C 180,E1 14048.265,E2 14048.265} C_VEL
LIN {X 0,Y 314.457,Z 989.03,A -85,B 0,C 180,E1 14056.313,E2 14056.313} C_VEL
LIN {X 0,Y 313.959,Z 989.596,A -85,B 0,C 180,E1 14063.172,E2 14063.172} C_VEL
LIN {X 0,Y 316.413,Z 994.787,A -85,B 0,C 180,E1 14064.91,E2 14064.91} C_VEL
LIN {X 0,Y 318.773,Z 997.683,A -85,B 0,C 180,E1 14066.303,E2 14066.303} C_VEL
LIN {X 0,Y 326.619,Z 1010.913,A -85,B 0,C 180,E1 14070.928,E2 14070.928} C_VEL
LIN {X 0,Y 337.643,Z 1033.06,A -85,B 0,C 180,E1 14077.292,E2 14077.292} C_VEL
LIN {X 0,Y 345.754,Z 1055.741,A -85,B 0,C 180,E1 14082.844,E2 14082.844} C_VEL
LIN {X 0,Y 350.799,Z 1078.421,A -85,B 0,C 180,E1 14087.957,E2 14087.957} C_VEL
LIN {X 0,Y 351.554,Z 1089.845,A -85,B 0,C 180,E1 14090.389,E2 14090.389} C_VEL
LIN {X 0,Y 341.252,Z 1117.959,A -85,B 0,C 180,E1 14095.297,E2 14095.297} C_VEL
LIN {X 0,Y 331.945,Z 1141.58,A -85,B 0,C 180,E1 14101.119,E2 14101.119} C_VEL
LIN {X 0,Y 324.888,Z 1159.594,A -85,B 0,C 180,E1 14107.47,E2 14107.47} C_VEL
LIN {X 0,Y 320.277,Z 1172.599,A -85,B 0,C 180,E1 14114.312,E2 14114.312} C_VEL
LIN {X 0,Y 318.257,Z 1179.864,A -85,B 0,C 180,E1 14120.448,E2 14120.448} C_VEL
LIN {X 0,Y 317.349,Z 1183.63,A -85,B 0,C 180,E1 14127.275,E2 14127.275} C_VEL
LIN {X 0,Y 317.373,Z 1183.435,A -85,B 0,C 180,E1 14133.202,E2 14133.202} C_VEL
LIN {X 0,Y 318.569,Z 1178.423,A -85,B 0,C 180,E1 14140.923,E2 14140.923} C_VEL
LIN {X 0,Y 321.868,Z 1167.873,A -85,B 0,C 180,E1 14148.45,E2 14148.45} C_VEL
LIN {X 0,Y 327.833,Z 1151.832,A -85,B 0,C 180,E1 14155.493,E2 14155.493} C_VEL
LIN {X 0,Y 336.233,Z 1130.806,A -85,B 0,C 180,E1 14161.696,E2 14161.696} C_VEL
LIN {X 0,Y 346.103,Z 1105.079,A -85,B 0,C 180,E1 14167.046,E2 14167.046} C_VEL
LIN {X 0,Y 351.881,Z 1087.977,A -85,B 0,C 180,E1 14169.827,E2 14169.827} C_VEL
LIN {X 0,Y 348.075,Z 1064.931,A -85,B 0,C 180,E1 14174.962,E2 14174.962} C_VEL
LIN {X 0,Y 340.824,Z 1040.953,A -85,B 0,C 180,E1 14180.569,E2 14180.569} C_VEL
LIN {X 0,Y 331.551,Z 1020.143,A -85,B 0,C 180,E1 14186.115,E2 14186.115} C_VEL
LIN {X 0,Y 321.801,Z 1002.424,A -85,B 0,C 180,E1 14191.751,E2 14191.751} C_VEL
LIN {X 0,Y 317.345,Z 995.542,A -85,B 0,C 180,E1 14194.421,E2 14194.421} C_VEL
LIN {X 0,Y 314.04,Z 990.386,A -85,B 0,C 180,E1 14196.514,E2 14196.514} C_VEL
LIN {X 0,Y 313.942,Z 989.03,A -85,B 0,C 180,E1 14196.747,E2 14196.747} C_VEL
LIN {X 0,Y 314.372,Z 989.03,A -85,B 0,C 180,E1 14203.747,E2 14203.747} C_VEL
LIN {X 0,Y 314.908,Z 989.03,A -85,B 0,C 180,E1 14211.735,E2 14211.735} C_VEL
LIN {X 0,Y 315.572,Z 989.03,A -85,B 0,C 180,E1 14220,E2 14220} C_VEL
LIN {X 0,Y 314.916,Z 989.03,A -85,B 0,C 180,E1 14228.265,E2 14228.265} C_VEL
LIN {X 0,Y 314.47,Z 989.03,A -85,B 0,C 180,E1 14236.314,E2 14236.314} C_VEL
LIN {X 0,Y 314.17,Z 989.371,A -85,B 0,C 180,E1 14239.972,E2 14239.972} C_VEL
LIN {X 0,Y 316.245,Z 994.442,A -85,B 0,C 180,E1 14241.216,E2 14241.216} C_VEL
LIN {X 0,Y 319.671,Z 997.596,A -85,B 0,C 180,E1 14242.827,E2 14242.827} C_VEL
LIN {X 0,Y 324.016,Z 1003.386,A -85,B 0,C 180,E1 14244.78,E2 14244.78} C_VEL
LIN {X 0,Y 339.044,Z 1025.974,A -85,B 0,C 180,E1 14250.635,E2 14250.635} C_VEL
LIN {X 0,Y 352.47,Z 1049.082,A -85,B 0,C 180,E1 14255.214,E2 14255.214} C_VEL
LIN {X 0,Y 366.031,Z 1079.54,A -85,B 0,C 180,E1 14259.908,E2 14259.908} C_VEL
LIN {X 0,Y 369.266,Z 1089.527,A -85,B 0,C 180,E1 14261.21,E2 14261.21} C_VEL
LIN {X 0,Y 360.153,Z 1127.968,A -85,B 0,C 180,E1 14263.605,E2 14263.605} C_VEL
LIN {X 0,Y 349.799,Z 1164.485,A -85,B 0,C 180,E1 14267.021,E2 14267.021} C_VEL
LIN {X 0,Y 339.243,Z 1198.079,A -85,B 0,C 180,E1 14271.482,E2 14271.482} C_VEL
LIN {X 0,Y 330.197,Z 1226.767,A -85,B 0,C 180,E1 14276.741,E2 14276.741} C_VEL
LIN {X 0,Y 323.01,Z 1251.931,A -85,B 0,C 180,E1 14283.04,E2 14283.04} C_VEL
LIN {X 0,Y 318.711,Z 1271.757,A -85,B 0,C 180,E1 14289.923,E2 14289.923} C_VEL
LIN {X 0,Y 317.112,Z 1284.478,A -85,B 0,C 180,E1 14296.235,E2 14296.235} C_VEL
LIN {X 0,Y 316.898,Z 1291.759,A -85,B 0,C 180,E1 14301.786,E2 14301.786} C_VEL
LIN {X 0,Y 317.101,Z 1295.621,A -85,B 0,C 180,E1 14307.855,E2 14307.855} C_VEL
LIN {X 0,Y 317.145,Z 1295.457,A -85,B 0,C 180,E1 14312.726,E2 14312.726} C_VEL
LIN {X 0,Y 316.852,Z 1291.759,A -85,B 0,C 180,E1 14318.213,E2 14318.213} C_VEL
LIN {X 0,Y 317.207,Z 1283.373,A -85,B 0,C 180,E1 14324.462,E2 14324.462} C_VEL
LIN {X 0,Y 319.281,Z 1268.319,A -85,B 0,C 180,E1 14331.486,E2 14331.486} C_VEL
LIN {X 0,Y 324.376,Z 1246.649,A -85,B 0,C 180,E1 14338.478,E2 14338.478} C_VEL
LIN {X 0,Y 332.32,Z 1219.905,A -85,B 0,C 180,E1 14344.681,E2 14344.681} C_VEL
LIN {X 0,Y 339.578,Z 1197.029,A -85,B 0,C 180,E1 14348.693,E2 14348.693} C_VEL
LIN {X 0,Y 340.137,Z 1184.845,A -85,B 0,C 180,E1 14350.822,E2 14350.822} C_VEL
LIN {X 0,Y 340.484,Z 1173.838,A -85,B 0,C 180,E1 14352.629,E2 14352.629} C_VEL
LIN {X 0,Y 340.987,Z 1172.15,A -85,B 0,C 180,E1 14352.85,E2 14352.85} C_VEL
LIN {X 0,Y 351.98,Z 1136.284,A -85,B 0,C 180,E1 14356.563,E2 14356.563} C_VEL
LIN {X 0,Y 362.18,Z 1096.951,A -85,B 0,C 180,E1 14359.282,E2 14359.282} C_VEL
LIN {X 0,Y 362.692,Z 1090.143,A -85,B 0,C 180,E1 14359.796,E2 14359.796} C_VEL
LIN {X 0,Y 350.695,Z 1060.128,A -85,B 0,C 180,E1 14364.415,E2 14364.415} C_VEL
LIN {X 0,Y 337.209,Z 1034.774,A -85,B 0,C 180,E1 14369.358,E2 14369.358} C_VEL
LIN {X 0,Y 324.433,Z 1015.347,A -85,B 0,C 180,E1 14374.449,E2 14374.449} C_VEL
LIN {X 0,Y 315.936,Z 1003.189,A -85,B 0,C 180,E1 14378.459,E2 14378.459} C_VEL
LIN {X 0,Y 312.097,Z 997.732,A -85,B 0,C 180,E1 14380.586,E2 14380.586} C_VEL
LIN {X 0,Y 306.812,Z 991.375,A -85,B 0,C 180,E1 14383.873,E2 14383.873} C_VEL
LIN {X 0,Y 306.459,Z 989.03,A -85,B 0,C 180,E1 14384.346,E2 14384.346} C_VEL
LIN {X 0,Y 306.898,Z 989.03,A -85,B 0,C 180,E1 14391.518,E2 14391.518} C_VEL
LIN {X 0,Y 307.448,Z 989.03,A -85,B 0,C 180,E1 14397.187,E2 14397.187} C_VEL
LIN {X 0,Y 307.403,Z 989.03,A -85,B 0,C 180,E1 14402.814,E2 14402.814} C_VEL
LIN {X 0,Y 306.816,Z 989.03,A -85,B 0,C 180,E1 14411.345,E2 14411.345} C_VEL
LIN {X 0,Y 306.288,Z 989.439,A -85,B 0,C 180,E1 14418.956,E2 14418.956} C_VEL
LIN {X 0,Y 308.755,Z 994.932,A -85,B 0,C 180,E1 14421.206,E2 14421.206} C_VEL
LIN {X 0,Y 311.215,Z 997.491,A -85,B 0,C 180,E1 14422.823,E2 14422.823} C_VEL
LIN {X 0,Y 315.036,Z 1003.152,A -85,B 0,C 180,E1 14425.439,E2 14425.439} C_VEL
LIN {X 0,Y 324.925,Z 1021.461,A -85,B 0,C 180,E1 14431.838,E2 14431.838} C_VEL
LIN {X 0,Y 334.349,Z 1042.854,A -85,B 0,C 180,E1 14437.945,E2 14437.945} C_VEL
LIN {X 0,Y 341.322,Z 1065.407,A -85,B 0,C 180,E1 14443.544,E2 14443.544} C_VEL
LIN {X 0,Y 345.129,Z 1087.521,A -85,B 0,C 180,E1 14448.702,E2 14448.702} C_VEL
LIN {X 0,Y 344.719,Z 1093.537,A -85,B 0,C 180,E1 14449.923,E2 14449.923} C_VEL
LIN {X 0,Y 334.253,Z 1120.825,A -85,B 0,C 180,E1 14454.859,E2 14454.859} C_VEL
LIN {X 0,Y 325.111,Z 1142.96,A -85,B 0,C 180,E1 14460.452,E2 14460.452} C_VEL
LIN {X 0,Y 317.646,Z 1160.978,A -85,B 0,C 180,E1 14466.927,E2 14466.927} C_VEL
LIN {X 0,Y 312.769,Z 1173.923,A -85,B 0,C 180,E1 14473.885,E2 14473.885} C_VEL
LIN {X 0,Y 310.564,Z 1181.24,A -85,B 0,C 180,E1 14480.21,E2 14480.21} C_VEL
LIN {X 0,Y 309.594,Z 1185,A -85,B 0,C 180,E1 14487.207,E2 14487.207} C_VEL
LIN {X 0,Y 309.649,Z 1184.955,A -85,B 0,C 180,E1 14492.794,E2 14492.794} C_VEL
LIN {X 0,Y 310.543,Z 1181.162,A -85,B 0,C 180,E1 14499.793,E2 14499.793} C_VEL
LIN {X 0,Y 313.569,Z 1171.648,A -85,B 0,C 180,E1 14507.505,E2 14507.505} C_VEL
LIN {X 0,Y 319.055,Z 1157.463,A -85,B 0,C 180,E1 14514.447,E2 14514.447} C_VEL
LIN {X 0,Y 327.091,Z 1138.201,A -85,B 0,C 180,E1 14520.815,E2 14520.815} C_VEL
LIN {X 0,Y 336.91,Z 1114.139,A -85,B 0,C 180,E1 14526.403,E2 14526.403} C_VEL
LIN {X 0,Y 345.37,Z 1090.529,A -85,B 0,C 180,E1 14530.518,E2 14530.518} C_VEL
LIN {X 0,Y 341.81,Z 1067.963,A -85,B 0,C 180,E1 14535.75,E2 14535.75} C_VEL
LIN {X 0,Y 335.21,Z 1045.085,A -85,B 0,C 180,E1 14541.349,E2 14541.349} C_VEL
LIN {X 0,Y 325.887,Z 1023.384,A -85,B 0,C 180,E1 14547.427,E2 14547.427} C_VEL
LIN {X 0,Y 317.862,Z 1008.78,A -85,B 0,C 180,E1 14552.429,E2 14552.429} C_VEL
LIN {X 0,Y 313.605,Z 1001.972,A -85,B 0,C 180,E1 14555.193,E2 14555.193} C_VEL
LIN {X 0,Y 310.052,Z 995.879,A -85,B 0,C 180,E1 14557.79,E2 14557.79} C_VEL
LIN {X 0,Y 306.476,Z 990.844,A -85,B 0,C 180,E1 14560.496,E2 14560.496} C_VEL
LIN {X 0,Y 306.264,Z 989.03,A -85,B 0,C 180,E1 14561.322,E2 14561.322} C_VEL
LIN {X 0,Y 306.686,Z 989.03,A -85,B 0,C 180,E1 14568.65,E2 14568.65} C_VEL
LIN {X 0,Y 307.464,Z 989.03,A -85,B 0,C 180,E1 14577.187,E2 14577.187} C_VEL
LIN {X 0,Y 307.418,Z 989.03,A -85,B 0,C 180,E1 14582.814,E2 14582.814} C_VEL
LIN {X 0,Y 306.825,Z 989.03,A -85,B 0,C 180,E1 14591.345,E2 14591.345} C_VEL
LIN {X 0,Y 306.591,Z 989.546,A -85,B 0,C 180,E1 14595.976,E2 14595.976} C_VEL
LIN {X 0,Y 308.766,Z 994.721,A -85,B 0,C 180,E1 14597.601,E2 14597.601} C_VEL
LIN {X 0,Y 312.097,Z 997.704,A -85,B 0,C 180,E1 14599.506,E2 14599.506} C_VEL
LIN {X 0,Y 316.173,Z 1003.339,A -85,B 0,C 180,E1 14601.73,E2 14601.73} C_VEL
LIN {X 0,Y 327.285,Z 1019.356,A -85,B 0,C 180,E1 14606.8,E2 14606.8} C_VEL
LIN {X 0,Y 340.78,Z 1040.954,A -85,B 0,C 180,E1 14612.013,E2 14612.013} C_VEL
LIN {X 0,Y 354.23,Z 1067.963,A -85,B 0,C 180,E1 14616.896,E2 14616.896} C_VEL
LIN {X 0,Y 363.07,Z 1092.398,A -85,B 0,C 180,E1 14620.481,E2 14620.481} C_VEL
LIN {X 0,Y 353.817,Z 1129.357,A -85,B 0,C 180,E1 14622.881,E2 14622.881} C_VEL
LIN {X 0,Y 343.021,Z 1165.575,A -85,B 0,C 180,E1 14626.378,E2 14626.378} C_VEL
LIN {X 0,Y 332.11,Z 1198.641,A -85,B 0,C 180,E1 14630.916,E2 14630.916} C_VEL
LIN {X 0,Y 322.471,Z 1227.742,A -85,B 0,C 180,E1 14636.466,E2 14636.466} C_VEL
LIN {X 0,Y 314.992,Z 1252.934,A -85,B 0,C 180,E1 14643.096,E2 14643.096} C_VEL
LIN {X 0,Y 310.492,Z 1273.108,A -85,B 0,C 180,E1 14650.621,E2 14650.621} C_VEL
LIN {X 0,Y 309.217,Z 1285.435,A -85,B 0,C 180,E1 14657.416,E2 14657.416} C_VEL
LIN {X 0,Y 309.182,Z 1292.666,A -85,B 0,C 180,E1 14664.397,E2 14664.397} C_VEL
LIN {X 0,Y 309.529,Z 1294.586,A -85,B 0,C 180,E1 14669.999,E2 14669.999} C_VEL
LIN {X 0,Y 309.178,Z 1292.672,A -85,B 0,C 180,E1 14675.601,E2 14675.601} C_VEL
LIN {X 0,Y 309.231,Z 1285.427,A -85,B 0,C 180,E1 14682.595,E2 14682.595} C_VEL
LIN {X 0,Y 310.693,Z 1272.04,A -85,B 0,C 180,E1 14689.875,E2 14689.875} C_VEL
LIN {X 0,Y 314.967,Z 1252.962,A -85,B 0,C 180,E1 14696.903,E2 14696.903} C_VEL
LIN {X 0,Y 322.325,Z 1228.007,A -85,B 0,C 180,E1 14703.489,E2 14703.489} C_VEL
LIN {X 0,Y 332.074,Z 1198.7,A -85,B 0,C 180,E1 14709.087,E2 14709.087} C_VEL
LIN {X 0,Y 340.987,Z 1172.15,A -85,B 0,C 180,E1 14712.85,E2 14712.85} C_VEL
LIN {X 0,Y 342.074,Z 1159.044,A -85,B 0,C 180,E1 14714.803,E2 14714.803} C_VEL
LIN {X 0,Y 342.704,Z 1147.118,A -85,B 0,C 180,E1 14716.421,E2 14716.421} C_VEL
LIN {X 0,Y 343.206,Z 1145.279,A -85,B 0,C 180,E1 14716.6,E2 14716.6} C_VEL
LIN {X 0,Y 354.129,Z 1106.772,A -85,B 0,C 180,E1 14719.612,E2 14719.612} C_VEL
LIN {X 0,Y 357.109,Z 1094.638,A -85,B 0,C 180,E1 14720.321,E2 14720.321} C_VEL
LIN {X 0,Y 345.827,Z 1064.976,A -85,B 0,C 180,E1 14725.062,E2 14725.062} C_VEL
LIN {X 0,Y 333.171,Z 1040.525,A -85,B 0,C 180,E1 14730.016,E2 14730.016} C_VEL
LIN {X 0,Y 320.872,Z 1021.115,A -85,B 0,C 180,E1 14735.288,E2 14735.288} C_VEL
LIN {X 0,Y 313.515,Z 1010.278,A -85,B 0,C 180,E1 14739.025,E2 14739.025} C_VEL
LIN {X 0,Y 308.686,Z 1003.552,A -85,B 0,C 180,E1 14741.843,E2 14741.843} C_VEL
LIN {X 0,Y 304.883,Z 998.515,A -85,B 0,C 180,E1 14744.424,E2 14744.424} C_VEL
LIN {X 0,Y 303.635,Z 996.397,A -85,B 0,C 180,E1 14745.42,E2 14745.42} C_VEL
LIN {X 0,Y 299.333,Z 991.891,A -85,B 0,C 180,E1 14749.171,E2 14749.171} C_VEL
LIN {X 0,Y 298.886,Z 989.03,A -85,B 0,C 180,E1 14750.357,E2 14750.357} C_VEL
LIN {X 0,Y 299.551,Z 989.03,A -85,B 0,C 180,E1 14757.113,E2 14757.113} C_VEL
LIN {X 0,Y 299.497,Z 989.03,A -85,B 0,C 180,E1 14762.888,E2 14762.888} C_VEL
LIN {X 0,Y 298.858,Z 989.03,A -85,B 0,C 180,E1 14771.652,E2 14771.652} C_VEL
LIN {X 0,Y 298.799,Z 989.971,A -85,B 0,C 180,E1 14773.414,E2 14773.414} C_VEL
LIN {X 0,Y 301.475,Z 995.219,A -85,B 0,C 180,E1 14776.645,E2 14776.645} C_VEL
LIN {X 0,Y 303.817,Z 997.395,A -85,B 0,C 180,E1 14778.648,E2 14778.648} C_VEL
LIN {X 0,Y 307.18,Z 1003.029,A -85,B 0,C 180,E1 14781.577,E2 14781.577} C_VEL
LIN {X 0,Y 312.625,Z 1012.358,A -85,B 0,C 180,E1 14785.747,E2 14785.747} C_VEL
LIN {X 0,Y 321.523,Z 1029.351,A -85,B 0,C 180,E1 14791.905,E2 14791.905} C_VEL
LIN {X 0,Y 330.129,Z 1050.779,A -85,B 0,C 180,E1 14798.167,E2 14798.167} C_VEL
LIN {X 0,Y 336.462,Z 1074.31,A -85,B 0,C 180,E1 14804.145,E2 14804.145} C_VEL
LIN {X 0,Y 338.862,Z 1094.693,A -85,B 0,C 180,E1 14809.038,E2 14809.038} C_VEL
LIN {X 0,Y 327.733,Z 1122.526,A -85,B 0,C 180,E1 14814.14,E2 14814.14} C_VEL
LIN {X 0,Y 317.812,Z 1145.449,A -85,B 0,C 180,E1 14820.097,E2 14820.097} C_VEL
LIN {X 0,Y 310.444,Z 1162.361,A -85,B 0,C 180,E1 14826.359,E2 14826.359} C_VEL
LIN {X 0,Y 305.618,Z 1174.308,A -85,B 0,C 180,E1 14832.768,E2 14832.768} C_VEL
LIN {X 0,Y 302.863,Z 1182.62,A -85,B 0,C 180,E1 14839.958,E2 14839.958} C_VEL
LIN {X 0,Y 301.843,Z 1186.369,A -85,B 0,C 180,E1 14847.135,E2 14847.135} C_VEL
LIN {X 0,Y 301.868,Z 1186.33,A -85,B 0,C 180,E1 14852.866,E2 14852.866} C_VEL
LIN {X 0,Y 302.844,Z 1182.542,A -85,B 0,C 180,E1 14860.045,E2 14860.045} C_VEL
LIN {X 0,Y 306.106,Z 1173.031,A -85,B 0,C 180,E1 14867.946,E2 14867.946} C_VEL
LIN {X 0,Y 311.927,Z 1158.85,A -85,B 0,C 180,E1 14875.044,E2 14875.044} C_VEL
LIN {X 0,Y 320.519,Z 1139.211,A -85,B 0,C 180,E1 14881.642,E2 14881.642} C_VEL
LIN {X 0,Y 331.031,Z 1114.537,A -85,B 0,C 180,E1 14887.404,E2 14887.404} C_VEL
LIN {X 0,Y 338.87,Z 1093.971,A -85,B 0,C 180,E1 14891.016,E2 14891.016} C_VEL
LIN {X 0,Y 335.868,Z 1072.178,A -85,B 0,C 180,E1 14896.279,E2 14896.279} C_VEL
LIN {X 0,Y 329.926,Z 1050.121,A -85,B 0,C 180,E1 14901.877,E2 14901.877} C_VEL
LIN {X 0,Y 321.369,Z 1028.688,A -85,B 0,C 180,E1 14908.114,E2 14908.114} C_VEL
LIN {X 0,Y 311.604,Z 1010.026,A -85,B 0,C 180,E1 14914.93,E2 14914.93} C_VEL
LIN {X 0,Y 306.706,Z 1002.682,A -85,B 0,C 180,E1 14918.548,E2 14918.548} C_VEL
LIN {X 0,Y 303.748,Z 997.143,A -85,B 0,C 180,E1 14921.218,E2 14921.218} C_VEL
LIN {X 0,Y 298.943,Z 991.196,A -85,B 0,C 180,E1 14925.941,E2 14925.941} C_VEL
LIN {X 0,Y 298.622,Z 989.03,A -85,B 0,C 180,E1 14926.857,E2 14926.857} C_VEL
LIN {X 0,Y 299.235,Z 989.03,A -85,B 0,C 180,E1 14934.212,E2 14934.212} C_VEL
LIN {X 0,Y 299.762,Z 989.03,A -85,B 0,C 180,E1 14940,E2 14940} C_VEL
LIN {X 0,Y 299.046,Z 989.03,A -85,B 0,C 180,E1 14948.707,E2 14948.707} C_VEL
LIN {X 0,Y 298.975,Z 989.684,A -85,B 0,C 180,E1 14950.413,E2 14950.413} C_VEL
LIN {X 0,Y 301.398,Z 994.917,A -85,B 0,C 180,E1 14953.02,E2 14953.02} C_VEL
LIN {X 0,Y 304.728,Z 997.683,A -85,B 0,C 180,E1 14955.529,E2 14955.529} C_VEL
LIN {X 0,Y 308.234,Z 1003.257,A -85,B 0,C 180,E1 14958.001,E2 14958.001} C_VEL
LIN {X 0,Y 310.306,Z 1005.88,A -85,B 0,C 180,E1 14959.254,E2 14959.254} C_VEL
LIN {X 0,Y 315.986,Z 1013.907,A -85,B 0,C 180,E1 14962.357,E2 14962.357} C_VEL
LIN {X 0,Y 324.823,Z 1027.036,A -85,B 0,C 180,E1 14966.549,E2 14966.549} C_VEL
LIN {X 0,Y 337.167,Z 1047.609,A -85,B 0,C 180,E1 14971.595,E2 14971.595} C_VEL
LIN {X 0,Y 349.428,Z 1073.536,A -85,B 0,C 180,E1 14976.425,E2 14976.425} C_VEL
LIN {X 0,Y 356.846,Z 1095.656,A -85,B 0,C 180,E1 14979.746,E2 14979.746} C_VEL
LIN {X 0,Y 346.035,Z 1135.846,A -85,B 0,C 180,E1 14982.551,E2 14982.551} C_VEL
LIN {X 0,Y 334.233,Z 1172.51,A -85,B 0,C 180,E1 14986.423,E2 14986.423} C_VEL
LIN {X 0,Y 322.945,Z 1204.907,A -85,B 0,C 180,E1 14991.319,E2 14991.319} C_VEL
LIN {X 0,Y 313.447,Z 1232.574,A -85,B 0,C 180,E1 14997.128,E2 14997.128} C_VEL
LIN {X 0,Y 306.49,Z 1255.37,A -85,B 0,C 180,E1 15003.696,E2 15003.696} C_VEL
LIN {X 0,Y 302.597,Z 1272.798,A -85,B 0,C 180,E1 15010.659,E2 15010.659} C_VEL
LIN {X 0,Y 301.405,Z 1284.021,A -85,B 0,C 180,E1 15017.085,E2 15017.085} C_VEL
LIN {X 0,Y 301.392,Z 1291.284,A -85,B 0,C 180,E1 15024.252,E2 15024.252} C_VEL
LIN {X 0,Y 301.761,Z 1293.215,A -85,B 0,C 180,E1 15029.999,E2 15029.999} C_VEL
LIN {X 0,Y 301.386,Z 1291.29,A -85,B 0,C 180,E1 15035.746,E2 15035.746} C_VEL
LIN {X 0,Y 301.422,Z 1284.015,A -85,B 0,C 180,E1 15042.927,E2 15042.927} C_VEL
LIN {X 0,Y 303.008,Z 1270.596,A -85,B 0,C 180,E1 15050.401,E2 15050.401} C_VEL
LIN {X 0,Y 307.673,Z 1251.229,A -85,B 0,C 180,E1 15057.685,E2 15057.685} C_VEL
LIN {X 0,Y 315.572,Z 1226.134,A -85,B 0,C 180,E1 15064.412,E2 15064.412} C_VEL
LIN {X 0,Y 325.678,Z 1197.24,A -85,B 0,C 180,E1 15070.006,E2 15070.006} C_VEL
LIN {X 0,Y 336.902,Z 1164.947,A -85,B 0,C 180,E1 15074.497,E2 15074.497} C_VEL
LIN {X 0,Y 343.206,Z 1145.279,A -85,B 0,C 180,E1 15076.6,E2 15076.6} C_VEL
LIN {X 0,Y 344.638,Z 1131.047,A -85,B 0,C 180,E1 15078.293,E2 15078.293} C_VEL
LIN {X 0,Y 345.901,Z 1116.424,A -85,B 0,C 180,E1 15079.884,E2 15079.884} C_VEL
LIN {X 0,Y 350.859,Z 1097.072,A -85,B 0,C 180,E1 15081.161,E2 15081.161} C_VEL
LIN {X 0,Y 340.976,Z 1070.124,A -85,B 0,C 180,E1 15085.651,E2 15085.651} C_VEL
LIN {X 0,Y 328.997,Z 1046.074,A -85,B 0,C 180,E1 15090.737,E2 15090.737} C_VEL
LIN {X 0,Y 316.105,Z 1024.49,A -85,B 0,C 180,E1 15096.787,E2 15096.787} C_VEL
LIN {X 0,Y 309.86,Z 1016.132,A -85,B 0,C 180,E1 15100.162,E2 15100.162} C_VEL
LIN {X 0,Y 306.265,Z 1010.703,A -85,B 0,C 180,E1 15102.494,E2 15102.494} C_VEL
LIN {X 0,Y 302.544,Z 1004.454,A -85,B 0,C 180,E1 15105.333,E2 15105.333} C_VEL
LIN {X 0,Y 297.718,Z 999.24,A -85,B 0,C 180,E1 15109.637,E2 15109.637} C_VEL
LIN {X 0,Y 297.044,Z 996.707,A -85,B 0,C 180,E1 15110.65,E2 15110.65} C_VEL
LIN {X 0,Y 292.508,Z 992.329,A -85,B 0,C 180,E1 15120,E2 15120} C_VEL
LIN {X 0,Y 293.61,Z 994.745,A -85,B 0,C 180,E1 15128.125,E2 15128.125} C_VEL
LIN {X 0,Y 296.741,Z 997.586,A -85,B 0,C 180,E1 15133.041,E2 15133.041} C_VEL
LIN {X 0,Y 299.637,Z 1002.952,A -85,B 0,C 180,E1 15136.701,E2 15136.701} C_VEL
LIN {X 0,Y 301.421,Z 1005.341,A -85,B 0,C 180,E1 15138.488,E2 15138.488} C_VEL
LIN {X 0,Y 305.41,Z 1012.084,A -85,B 0,C 180,E1 15142.131,E2 15142.131} C_VEL
LIN {X 0,Y 312.321,Z 1025.227,A -85,B 0,C 180,E1 15147.774,E2 15147.774} C_VEL
LIN {X 0,Y 320.486,Z 1043.485,A -85,B 0,C 180,E1 15154.013,E2 15154.013} C_VEL
LIN {X 0,Y 327.285,Z 1064.312,A -85,B 0,C 180,E1 15159.939,E2 15159.939} C_VEL
LIN {X 0,Y 331.516,Z 1085.598,A -85,B 0,C 180,E1 15165.416,E2 15165.416} C_VEL
LIN {X 0,Y 332.213,Z 1098.054,A -85,B 0,C 180,E1 15168.472,E2 15168.472} C_VEL
LIN {X 0,Y 321.142,Z 1124.539,A -85,B 0,C 180,E1 15173.463,E2 15173.463} C_VEL
LIN {X 0,Y 311.027,Z 1146.833,A -85,B 0,C 180,E1 15179.375,E2 15179.375} C_VEL
LIN {X 0,Y 303.261,Z 1163.747,A -85,B 0,C 180,E1 15185.764,E2 15185.764} C_VEL
LIN {X 0,Y 297.675,Z 1176.806,A -85,B 0,C 180,E1 15193.13,E2 15193.13} C_VEL
LIN {X 0,Y 295.175,Z 1183.997,A -85,B 0,C 180,E1 15199.694,E2 15199.694} C_VEL
LIN {X 0,Y 294.079,Z 1187.74,A -85,B 0,C 180,E1 15207.06,E2 15207.06} C_VEL
LIN {X 0,Y 294.104,Z 1187.703,A -85,B 0,C 180,E1 15212.942,E2 15212.942} C_VEL
LIN {X 0,Y 295.158,Z 1183.921,A -85,B 0,C 180,E1 15220.309,E2 15220.309} C_VEL
LIN {X 0,Y 298.643,Z 1174.419,A -85,B 0,C 180,E1 15228.411,E2 15228.411} C_VEL
LIN {X 0,Y 304.809,Z 1160.241,A -85,B 0,C 180,E1 15235.671,E2 15235.671} C_VEL
LIN {X 0,Y 313.704,Z 1140.937,A -85,B 0,C 180,E1 15242.3,E2 15242.3} C_VEL
LIN {X 0,Y 324.429,Z 1116.911,A -85,B 0,C 180,E1 15248.046,E2 15248.046} C_VEL
LIN {X 0,Y 332.379,Z 1096.964,A -85,B 0,C 180,E1 15251.642,E2 15251.642} C_VEL
LIN {X 0,Y 329.708,Z 1075.421,A -85,B 0,C 180,E1 15257.08,E2 15257.08} C_VEL
LIN {X 0,Y 324.257,Z 1053.895,A -85,B 0,C 180,E1 15262.774,E2 15262.774} C_VEL
LIN {X 0,Y 316.606,Z 1034.058,A -85,B 0,C 180,E1 15268.855,E2 15268.855} C_VEL
LIN {X 0,Y 308.143,Z 1016.814,A -85,B 0,C 180,E1 15275.403,E2 15275.403} C_VEL
LIN {X 0,Y 303.548,Z 1009.555,A -85,B 0,C 180,E1 15279.161,E2 15279.161} C_VEL
LIN {X 0,Y 300.307,Z 1003.486,A -85,B 0,C 180,E1 15282.454,E2 15282.454} C_VEL
LIN {X 0,Y 296.788,Z 998.405,A -85,B 0,C 180,E1 15286.4,E2 15286.4} C_VEL
LIN {X 0,Y 295.885,Z 996.421,A -85,B 0,C 180,E1 15287.856,E2 15287.856} C_VEL
LIN {X 0,Y 292.216,Z 991.918,A -85,B 0,C 180,E1 15297.04,E2 15297.04} C_VEL
LIN {X 0,Y 292.586,Z 992.777,A -85,B 0,C 180,E1 15301.847,E2 15301.847} C_VEL
LIN {X 0,Y 297.357,Z 997.482,A -85,B 0,C 180,E1 15309.99,E2 15309.99} C_VEL
LIN {X 0,Y 300.484,Z 1003.026,A -85,B 0,C 180,E1 15313.245,E2 15313.245} C_VEL
LIN {X 0,Y 302.889,Z 1005.347,A -85,B 0,C 180,E1 15315.111,E2 15315.111} C_VEL
LIN {X 0,Y 306.763,Z 1011.026,A -85,B 0,C 180,E1 15317.905,E2 15317.905} C_VEL
LIN {X 0,Y 314.101,Z 1022.11,A -85,B 0,C 180,E1 15322.292,E2 15322.292} C_VEL
LIN {X 0,Y 324.667,Z 1038.488,A -85,B 0,C 180,E1 15327.411,E2 15327.411} C_VEL
LIN {X 0,Y 337.358,Z 1062.168,A -85,B 0,C 180,E1 15332.843,E2 15332.843} C_VEL
LIN {X 0,Y 348.63,Z 1090.243,A -85,B 0,C 180,E1 15337.798,E2 15337.798} C_VEL
LIN {X 0,Y 350.716,Z 1098.411,A -85,B 0,C 180,E1 15338.976,E2 15338.976} C_VEL
LIN {X 0,Y 340.246,Z 1135.374,A -85,B 0,C 180,E1 15341.626,E2 15341.626} C_VEL
LIN {X 0,Y 328.182,Z 1171.414,A -85,B 0,C 180,E1 15345.478,E2 15345.478} C_VEL
LIN {X 0,Y 316.745,Z 1202.836,A -85,B 0,C 180,E1 15350.271,E2 15350.271} C_VEL
LIN {X 0,Y 306.36,Z 1231.368,A -85,B 0,C 180,E1 15356.348,E2 15356.348} C_VEL
LIN {X 0,Y 299.074,Z 1253.904,A -85,B 0,C 180,E1 15362.991,E2 15362.991} C_VEL
LIN {X 0,Y 294.957,Z 1271.138,A -85,B 0,C 180,E1 15370.025,E2 15370.025} C_VEL
LIN {X 0,Y 293.53,Z 1283.727,A -85,B 0,C 180,E1 15377.615,E2 15377.615} C_VEL
LIN {X 0,Y 293.588,Z 1289.899,A -85,B 0,C 180,E1 15384.099,E2 15384.099} C_VEL
LIN {X 0,Y 293.997,Z 1291.845,A -85,B 0,C 180,E1 15389.999,E2 15389.999} C_VEL
LIN {X 0,Y 293.58,Z 1289.906,A -85,B 0,C 180,E1 15395.899,E2 15395.899} C_VEL
LIN {X 0,Y 293.528,Z 1283.739,A -85,B 0,C 180,E1 15402.383,E2 15402.383} C_VEL
LIN {X 0,Y 294.623,Z 1273.008,A -85,B 0,C 180,E1 15409.047,E2 15409.047} C_VEL
LIN {X 0,Y 298.734,Z 1255.007,A -85,B 0,C 180,E1 15416.634,E2 15416.634} C_VEL
LIN {X 0,Y 305.88,Z 1232.853,A -85,B 0,C 180,E1 15423.286,E2 15423.286} C_VEL
LIN {X 0,Y 316.146,Z 1204.474,A -85,B 0,C 180,E1 15429.442,E2 15429.442} C_VEL
LIN {X 0,Y 327.792,Z 1172.868,A -85,B 0,C 180,E1 15434.331,E2 15434.331} C_VEL
LIN {X 0,Y 339.247,Z 1138.819,A -85,B 0,C 180,E1 15438.064,E2 15438.064} C_VEL
LIN {X 0,Y 345.901,Z 1116.424,A -85,B 0,C 180,E1 15439.884,E2 15439.884} C_VEL
LIN {X 0,Y 346.481,Z 1105.374,A -85,B 0,C 180,E1 15441.054,E2 15441.054} C_VEL
LIN {X 0,Y 341.465,Z 1089.605,A -85,B 0,C 180,E1 15443.658,E2 15443.658} C_VEL
LIN {X 0,Y 330.706,Z 1063.049,A -85,B 0,C 180,E1 15448.734,E2 15448.734} C_VEL
LIN {X 0,Y 318.319,Z 1040.202,A -85,B 0,C 180,E1 15454.544,E2 15454.544} C_VEL
LIN {X 0,Y 308.685,Z 1024.685,A -85,B 0,C 180,E1 15459.879,E2 15459.879} C_VEL
LIN {X 0,Y 303.712,Z 1017.736,A -85,B 0,C 180,E1 15463.1,E2 15463.1} C_VEL
LIN {X 0,Y 299.695,Z 1011.389,A -85,B 0,C 180,E1 15466.349,E2 15466.349} C_VEL
LIN {X 0,Y 295.735,Z 1005.954,A -85,B 0,C 180,E1 15470.363,E2 15470.363} C_VEL
LIN {X 0,Y 294.898,Z 1004.22,A -85,B 0,C 180,E1 15471.541,E2 15471.541} C_VEL
LIN {X 0,Y 291.022,Z 1000.118,A -85,B 0,C 180,E1 15480,E2 15480} C_VEL
LIN {X 0,Y 291.939,Z 1002.511,A -85,B 0,C 180,E1 15488.172,E2 15488.172} C_VEL
LIN {X 0,Y 294.594,Z 1005.226,A -85,B 0,C 180,E1 15492.743,E2 15492.743} C_VEL
LIN {X 0,Y 297.656,Z 1010.722,A -85,B 0,C 180,E1 15496.924,E2 15496.924} C_VEL
LIN {X 0,Y 302.416,Z 1019.718,A -85,B 0,C 180,E1 15501.976,E2 15501.976} C_VEL
LIN {X 0,Y 308.486,Z 1031.606,A -85,B 0,C 180,E1 15507.296,E2 15507.296} C_VEL
LIN {X 0,Y 316.008,Z 1049.795,A -85,B 0,C 180,E1 15513.717,E2 15513.717} C_VEL
LIN {X 0,Y 321.937,Z 1070.113,A -85,B 0,C 180,E1 15519.689,E2 15519.689} C_VEL
LIN {X 0,Y 325.415,Z 1090.766,A -85,B 0,C 180,E1 15525.223,E2 15525.223} C_VEL
LIN {X 0,Y 325.767,Z 1101.046,A -85,B 0,C 180,E1 15527.826,E2 15527.826} C_VEL
LIN {X 0,Y 313.549,Z 1128.879,A -85,B 0,C 180,E1 15533.286,E2 15533.286} C_VEL
LIN {X 0,Y 302.753,Z 1151.498,A -85,B 0,C 180,E1 15539.692,E2 15539.692} C_VEL
LIN {X 0,Y 294.346,Z 1168.882,A -85,B 0,C 180,E1 15546.961,E2 15546.961} C_VEL
LIN {X 0,Y 289.062,Z 1180.943,A -85,B 0,C 180,E1 15554.871,E2 15554.871} C_VEL
LIN {X 0,Y 287.05,Z 1186.43,A -85,B 0,C 180,E1 15560.927,E2 15560.927} C_VEL
LIN {X 0,Y 286.329,Z 1189.11,A -85,B 0,C 180,E1 15566.98,E2 15566.98} C_VEL
LIN {X 0,Y 286.345,Z 1189.074,A -85,B 0,C 180,E1 15573.022,E2 15573.022} C_VEL
LIN {X 0,Y 287.465,Z 1185.302,A -85,B 0,C 180,E1 15580.588,E2 15580.588} C_VEL
LIN {X 0,Y 291.202,Z 1175.806,A -85,B 0,C 180,E1 15588.899,E2 15588.899} C_VEL
LIN {X 0,Y 297.733,Z 1161.632,A -85,B 0,C 180,E1 15596.327,E2 15596.327} C_VEL
LIN {X 0,Y 307.265,Z 1141.948,A -85,B 0,C 180,E1 15603.192,E2 15603.192} C_VEL
LIN {X 0,Y 318.318,Z 1118.285,A -85,B 0,C 180,E1 15608.913,E2 15608.913} C_VEL
LIN {X 0,Y 325.936,Z 1100.294,A -85,B 0,C 180,E1 15612.206,E2 15612.206} C_VEL
LIN {X 0,Y 323.714,Z 1079.381,A -85,B 0,C 180,E1 15617.696,E2 15617.696} C_VEL
LIN {X 0,Y 318.783,Z 1058.099,A -85,B 0,C 180,E1 15623.585,E2 15623.585} C_VEL
LIN {X 0,Y 311.987,Z 1039.595,A -85,B 0,C 180,E1 15629.554,E2 15629.554} C_VEL
LIN {X 0,Y 304.786,Z 1023.702,A -85,B 0,C 180,E1 15635.796,E2 15635.796} C_VEL
LIN {X 0,Y 297.504,Z 1010.667,A -85,B 0,C 180,E1 15642.955,E2 15642.955} C_VEL
LIN {X 0,Y 294.532,Z 1005.398,A -85,B 0,C 180,E1 15646.955,E2 15646.955} C_VEL
LIN {X 0,Y 293.003,Z 1003.574,A -85,B 0,C 180,E1 15649.267,E2 15649.267} C_VEL
LIN {X 0,Y 290.72,Z 999.703,A -85,B 0,C 180,E1 15657.025,E2 15657.025} C_VEL
LIN {X 0,Y 291.253,Z 1000.752,A -85,B 0,C 180,E1 15662.227,E2 15662.227} C_VEL
LIN {X 0,Y 295.663,Z 1005.345,A -85,B 0,C 180,E1 15669.666,E2 15669.666} C_VEL
LIN {X 0,Y 299.093,Z 1010.868,A -85,B 0,C 180,E1 15673.308,E2 15673.308} C_VEL
LIN {X 0,Y 300.996,Z 1013.453,A -85,B 0,C 180,E1 15674.911,E2 15674.911} C_VEL
LIN {X 0,Y 306.182,Z 1021.301,A -85,B 0,C 180,E1 15678.678,E2 15678.678} C_VEL
LIN {X 0,Y 313.748,Z 1032.473,A -85,B 0,C 180,E1 15683.125,E2 15683.125} C_VEL
LIN {X 0,Y 325.724,Z 1053.201,A -85,B 0,C 180,E1 15689.049,E2 15689.049} C_VEL
LIN {X 0,Y 336.681,Z 1076.922,A -85,B 0,C 180,E1 15694.072,E2 15694.072} C_VEL
LIN {X 0,Y 344.64,Z 1099.648,A -85,B 0,C 180,E1 15698.033,E2 15698.033} C_VEL
LIN {X 0,Y 333.675,Z 1137.621,A -85,B 0,C 180,E1 15700.919,E2 15700.919} C_VEL
LIN {X 0,Y 321.514,Z 1172.218,A -85,B 0,C 180,E1 15704.748,E2 15704.748} C_VEL
LIN {X 0,Y 309.653,Z 1203.272,A -85,B 0,C 180,E1 15709.642,E2 15709.642} C_VEL
LIN {X 0,Y 298.926,Z 1231.33,A -85,B 0,C 180,E1 15715.832,E2 15715.832} C_VEL
LIN {X 0,Y 291.049,Z 1254.594,A -85,B 0,C 180,E1 15723.02,E2 15723.02} C_VEL
LIN {X 0,Y 286.773,Z 1272.289,A -85,B 0,C 180,E1 15730.8,E2 15730.8} C_VEL
LIN {X 0,Y 285.688,Z 1282.944,A -85,B 0,C 180,E1 15737.801,E2 15737.801} C_VEL
LIN {X 0,Y 285.77,Z 1288.512,A -85,B 0,C 180,E1 15743.937,E2 15743.937} C_VEL
LIN {X 0,Y 286.21,Z 1290.471,A -85,B 0,C 180,E1 15749.999,E2 15749.999} C_VEL
LIN {X 0,Y 285.76,Z 1288.519,A -85,B 0,C 180,E1 15756.061,E2 15756.061} C_VEL
LIN {X 0,Y 285.684,Z 1282.957,A -85,B 0,C 180,E1 15762.197,E2 15762.197} C_VEL
LIN {X 0,Y 286.785,Z 1272.421,A -85,B 0,C 180,E1 15769.141,E2 15769.141} C_VEL
LIN {X 0,Y 291.021,Z 1254.623,A -85,B 0,C 180,E1 15776.981,E2 15776.981} C_VEL
LIN {X 0,Y 298.865,Z 1231.367,A -85,B 0,C 180,E1 15784.173,E2 15784.173} C_VEL
LIN {X 0,Y 309.639,Z 1203.357,A -85,B 0,C 180,E1 15790.354,E2 15790.354} C_VEL
LIN {X 0,Y 321.849,Z 1171.74,A -85,B 0,C 180,E1 15795.311,E2 15795.311} C_VEL
LIN {X 0,Y 333.489,Z 1138.534,A -85,B 0,C 180,E1 15798.998,E2 15798.998} C_VEL
LIN {X 0,Y 344.47,Z 1101.804,A -85,B 0,C 180,E1 15801.787,E2 15801.787} C_VEL
LIN {X 0,Y 343.377,Z 1095.3,A -85,B 0,C 180,E1 15802.699,E2 15802.699} C_VEL
LIN {X 0,Y 341.465,Z 1089.605,A -85,B 0,C 180,E1 15803.658,E2 15803.658} C_VEL
LIN {X 0,Y 336.72,Z 1082.659,A -85,B 0,C 180,E1 15805.363,E2 15805.363} C_VEL
LIN {X 0,Y 328.002,Z 1072.687,A -85,B 0,C 180,E1 15808.42,E2 15808.42} C_VEL
LIN {X 0,Y 316.163,Z 1048.963,A -85,B 0,C 180,E1 15814.357,E2 15814.357} C_VEL
LIN {X 0,Y 306.115,Z 1031.968,A -85,B 0,C 180,E1 15820.191,E2 15820.191} C_VEL
LIN {X 0,Y 300.792,Z 1024.446,A -85,B 0,C 180,E1 15823.875,E2 15823.875} C_VEL
LIN {X 0,Y 297.48,Z 1018.786,A -85,B 0,C 180,E1 15826.829,E2 15826.829} C_VEL
LIN {X 0,Y 293.745,Z 1012.938,A -85,B 0,C 180,E1 15830.968,E2 15830.968} C_VEL
LIN {X 0,Y 289.426,Z 1007.885,A -85,B 0,C 180,E1 15840,E2 15840} C_VEL
LIN {X 0,Y 290.034,Z 1010.136,A -85,B 0,C 180,E1 15848.037,E2 15848.037} C_VEL
LIN {X 0,Y 292.284,Z 1012.76,A -85,B 0,C 180,E1 15852.497,E2 15852.497} C_VEL
LIN {X 0,Y 294.775,Z 1017.877,A -85,B 0,C 180,E1 15856.352,E2 15856.352} C_VEL
LIN {X 0,Y 299.287,Z 1026.888,A -85,B 0,C 180,E1 15861.703,E2 15861.703} C_VEL
LIN {X 0,Y 304.829,Z 1038.985,A -85,B 0,C 180,E1 15867.227,E2 15867.227} C_VEL
LIN {X 0,Y 311.414,Z 1056.383,A -85,B 0,C 180,E1 15873.543,E2 15873.543} C_VEL
LIN {X 0,Y 316.569,Z 1076.262,A -85,B 0,C 180,E1 15879.57,E2 15879.57} C_VEL
LIN {X 0,Y 319.353,Z 1096.348,A -85,B 0,C 180,E1 15885.133,E2 15885.133} C_VEL
LIN {X 0,Y 319.055,Z 1104.832,A -85,B 0,C 180,E1 15887.29,E2 15887.29} C_VEL
LIN {X 0,Y 306.187,Z 1132.546,A -85,B 0,C 180,E1 15892.974,E2 15892.974} C_VEL
LIN {X 0,Y 295.455,Z 1153.876,A -85,B 0,C 180,E1 15899.288,E2 15899.288} C_VEL
LIN {X 0,Y 287.355,Z 1169.862,A -85,B 0,C 180,E1 15906.126,E2 15906.126} C_VEL
LIN {X 0,Y 281.507,Z 1182.324,A -85,B 0,C 180,E1 15914.454,E2 15914.454} C_VEL
LIN {X 0,Y 279.342,Z 1187.808,A -85,B 0,C 180,E1 15920.675,E2 15920.675} C_VEL
LIN {X 0,Y 278.565,Z 1190.482,A -85,B 0,C 180,E1 15926.896,E2 15926.896} C_VEL
LIN {X 0,Y 278.58,Z 1190.446,A -85,B 0,C 180,E1 15933.106,E2 15933.106} C_VEL
LIN {X 0,Y 279.777,Z 1186.683,A -85,B 0,C 180,E1 15940.883,E2 15940.883} C_VEL
LIN {X 0,Y 283.801,Z 1177.19,A -85,B 0,C 180,E1 15949.411,E2 15949.411} C_VEL
LIN {X 0,Y 290.7,Z 1163.023,A -85,B 0,C 180,E1 15957.015,E2 15957.015} C_VEL
LIN {X 0,Y 300.763,Z 1143.295,A -85,B 0,C 180,E1 15964.019,E2 15964.019} C_VEL
LIN {X 0,Y 312.279,Z 1119.667,A -85,B 0,C 180,E1 15969.814,E2 15969.814} C_VEL
LIN {X 0,Y 319.515,Z 1103.072,A -85,B 0,C 180,E1 15972.939,E2 15972.939} C_VEL
LIN {X 0,Y 317.556,Z 1082.186,A -85,B 0,C 180,E1 15978.65,E2 15978.65} C_VEL
LIN {X 0,Y 313.442,Z 1062.836,A -85,B 0,C 180,E1 15984.253,E2 15984.253} C_VEL
LIN {X 0,Y 307.046,Z 1044.215,A -85,B 0,C 180,E1 15990.565,E2 15990.565} C_VEL
LIN {X 0,Y 301.016,Z 1030.212,A -85,B 0,C 180,E1 15996.358,E2 15996.358} C_VEL
LIN {X 0,Y 295.74,Z 1019.492,A -85,B 0,C 180,E1 16002.174,E2 16002.174} C_VEL
LIN {X 0,Y 292.1,Z 1012.343,A -85,B 0,C 180,E1 16007.508,E2 16007.508} C_VEL
LIN {X 0,Y 289.019,Z 1007.484,A -85,B 0,C 180,E1 16017.007,E2 16017.007} C_VEL
LIN {X 0,Y 289.785,Z 1008.599,A -85,B 0,C 180,E1 16022.425,E2 16022.425} C_VEL
LIN {X 0,Y 293.83,Z 1012.965,A -85,B 0,C 180,E1 16029.342,E2 16029.342} C_VEL
LIN {X 0,Y 297.59,Z 1018.711,A -85,B 0,C 180,E1 16033.376,E2 16033.376} C_VEL
LIN {X 0,Y 304.085,Z 1029.301,A -85,B 0,C 180,E1 16038.612,E2 16038.612} C_VEL
LIN {X 0,Y 311.024,Z 1039.922,A -85,B 0,C 180,E1 16042.838,E2 16042.838} C_VEL
LIN {X 0,Y 322.127,Z 1060.002,A -85,B 0,C 180,E1 16048.695,E2 16048.695} C_VEL
LIN {X 0,Y 332.428,Z 1084.035,A -85,B 0,C 180,E1 16053.893,E2 16053.893} C_VEL
LIN {X 0,Y 338.648,Z 1102.953,A -85,B 0,C 180,E1 16057.287,E2 16057.287} C_VEL
LIN {X 0,Y 326.312,Z 1142.507,A -85,B 0,C 180,E1 16060.443,E2 16060.443} C_VEL
LIN {X 0,Y 312.986,Z 1177.902,A -85,B 0,C 180,E1 16064.67,E2 16064.67} C_VEL
LIN {X 0,Y 300.595,Z 1208.641,A -85,B 0,C 180,E1 16069.965,E2 16069.965} C_VEL
LIN {X 0,Y 290.125,Z 1234.962,A -85,B 0,C 180,E1 16076.322,E2 16076.322} C_VEL
LIN {X 0,Y 282.511,Z 1257.178,A -85,B 0,C 180,E1 16083.852,E2 16083.852} C_VEL
LIN {X 0,Y 278.576,Z 1273.615,A -85,B 0,C 180,E1 16091.86,E2 16091.86} C_VEL
LIN {X 0,Y 277.833,Z 1283.505,A -85,B 0,C 180,E1 16099.222,E2 16099.222} C_VEL
LIN {X 0,Y 277.961,Z 1287.125,A -85,B 0,C 180,E1 16103.766,E2 16103.766} C_VEL
LIN {X 0,Y 278.446,Z 1289.101,A -85,B 0,C 180,E1 16109.999,E2 16109.999} C_VEL
LIN {X 0,Y 277.949,Z 1287.132,A -85,B 0,C 180,E1 16116.232,E2 16116.232} C_VEL
LIN {X 0,Y 277.841,Z 1281.54,A -85,B 0,C 180,E1 16122.546,E2 16122.546} C_VEL
LIN {X 0,Y 279.071,Z 1270.865,A -85,B 0,C 180,E1 16129.751,E2 16129.751} C_VEL
LIN {X 0,Y 283.687,Z 1253.167,A -85,B 0,C 180,E1 16137.737,E2 16137.737} C_VEL
LIN {X 0,Y 292.024,Z 1229.901,A -85,B 0,C 180,E1 16145.09,E2 16145.09} C_VEL
LIN {X 0,Y 303.238,Z 1202.185,A -85,B 0,C 180,E1 16151.316,E2 16151.316} C_VEL
LIN {X 0,Y 316.087,Z 1170.284,A -85,B 0,C 180,E1 16156.377,E2 16156.377} C_VEL
LIN {X 0,Y 328.075,Z 1137.467,A -85,B 0,C 180,E1 16160.039,E2 16160.039} C_VEL
LIN {X 0,Y 338.577,Z 1102.408,A -85,B 0,C 180,E1 16162.813,E2 16162.813} C_VEL
LIN {X 0,Y 329.258,Z 1075.624,A -85,B 0,C 180,E1 16167.808,E2 16167.808} C_VEL
LIN {X 0,Y 328.002,Z 1072.687,A -85,B 0,C 180,E1 16168.42,E2 16168.42} C_VEL
LIN {X 0,Y 323.147,Z 1066.859,A -85,B 0,C 180,E1 16170.303,E2 16170.303} C_VEL
LIN {X 0,Y 314.507,Z 1059.361,A -85,B 0,C 180,E1 16173.721,E2 16173.721} C_VEL
LIN {X 0,Y 305.068,Z 1042.303,A -85,B 0,C 180,E1 16179.35,E2 16179.35} C_VEL
LIN {X 0,Y 298.523,Z 1031.907,A -85,B 0,C 180,E1 16184.095,E2 16184.095} C_VEL
LIN {X 0,Y 294.946,Z 1026.027,A -85,B 0,C 180,E1 16187.348,E2 16187.348} C_VEL
LIN {X 0,Y 291.021,Z 1019.452,A -85,B 0,C 180,E1 16192.177,E2 16192.177} C_VEL
LIN {X 0,Y 287.581,Z 1015.577,A -85,B 0,C 180,E1 16200,E2 16200} C_VEL
LIN {X 0,Y 288.007,Z 1017.884,A -85,B 0,C 180,E1 16208.331,E2 16208.331} C_VEL
LIN {X 0,Y 289.815,Z 1019.853,A -85,B 0,C 180,E1 16212.021,E2 16212.021} C_VEL
LIN {X 0,Y 293.277,Z 1028.096,A -85,B 0,C 180,E1 16217.981,E2 16217.981} C_VEL
LIN {X 0,Y 298.784,Z 1040.343,A -85,B 0,C 180,E1 16224.622,E2 16224.622} C_VEL
LIN {X 0,Y 304.25,Z 1054.719,A -85,B 0,C 180,E1 16230.476,E2 16230.476} C_VEL
LIN {X 0,Y 309.563,Z 1073.729,A -85,B 0,C 180,E1 16236.868,E2 16236.868} C_VEL
LIN {X 0,Y 312.677,Z 1093.932,A -85,B 0,C 180,E1 16242.844,E2 16242.844} C_VEL
LIN {X 0,Y 312.862,Z 1107.322,A -85,B 0,C 180,E1 16246.514,E2 16246.514} C_VEL
LIN {X 0,Y 299.749,Z 1134.341,A -85,B 0,C 180,E1 16252.18,E2 16252.18} C_VEL
LIN {X 0,Y 288.738,Z 1155.259,A -85,B 0,C 180,E1 16258.493,E2 16258.493} C_VEL
LIN {X 0,Y 279.703,Z 1172.153,A -85,B 0,C 180,E1 16265.991,E2 16265.991} C_VEL
LIN {X 0,Y 273.969,Z 1183.706,A -85,B 0,C 180,E1 16274.015,E2 16274.015} C_VEL
LIN {X 0,Y 271.644,Z 1189.184,A -85,B 0,C 180,E1 16280.408,E2 16280.408} C_VEL
LIN {X 0,Y 270.812,Z 1191.852,A -85,B 0,C 180,E1 16286.807,E2 16286.807} C_VEL
LIN {X 0,Y 270.823,Z 1191.817,A -85,B 0,C 180,E1 16293.195,E2 16293.195} C_VEL
LIN {X 0,Y 272.11,Z 1188.062,A -85,B 0,C 180,E1 16301.193,E2 16301.193} C_VEL
LIN {X 0,Y 276.428,Z 1178.572,A -85,B 0,C 180,E1 16309.95,E2 16309.95} C_VEL
LIN {X 0,Y 283.714,Z 1164.412,A -85,B 0,C 180,E1 16317.737,E2 16317.737} C_VEL
LIN {X 0,Y 294.356,Z 1144.595,A -85,B 0,C 180,E1 16324.895,E2 16324.895} C_VEL
LIN {X 0,Y 306.31,Z 1121.05,A -85,B 0,C 180,E1 16330.751,E2 16330.751} C_VEL
LIN {X 0,Y 313.134,Z 1105.827,A -85,B 0,C 180,E1 16333.712,E2 16333.712} C_VEL
LIN {X 0,Y 311.6,Z 1086.149,A -85,B 0,C 180,E1 16339.319,E2 16339.319} C_VEL
LIN {X 0,Y 307.849,Z 1066.566,A -85,B 0,C 180,E1 16345.244,E2 16345.244} C_VEL
LIN {X 0,Y 302.126,Z 1048.478,A -85,B 0,C 180,E1 16351.675,E2 16351.675} C_VEL
LIN {X 0,Y 295.438,Z 1032.48,A -85,B 0,C 180,E1 16359.052,E2 16359.052} C_VEL
LIN {X 0,Y 292.023,Z 1025.445,A -85,B 0,C 180,E1 16363.489,E2 16363.489} C_VEL
LIN {X 0,Y 289.196,Z 1018.991,A -85,B 0,C 180,E1 16368.717,E2 16368.717} C_VEL
LIN {X 0,Y 287.169,Z 1015.214,A -85,B 0,C 180,E1 16376.988,E2 16376.988} C_VEL
LIN {X 0,Y 287.879,Z 1016.225,A -85,B 0,C 180,E1 16382.253,E2 16382.253} C_VEL
LIN {X 0,Y 291.773,Z 1020.694,A -85,B 0,C 180,E1 16389.128,E2 16389.128} C_VEL
LIN {X 0,Y 296.514,Z 1028.445,A -85,B 0,C 180,E1 16394.27,E2 16394.27} C_VEL
LIN {X 0,Y 304.232,Z 1040.557,A -85,B 0,C 180,E1 16400.126,E2 16400.126} C_VEL
LIN {X 0,Y 314.551,Z 1059.334,A -85,B 0,C 180,E1 16406.342,E2 16406.342} C_VEL
LIN {X 0,Y 324.876,Z 1082.324,A -85,B 0,C 180,E1 16411.945,E2 16411.945} C_VEL
LIN {X 0,Y 332.458,Z 1105.386,A -85,B 0,C 180,E1 16416.379,E2 16416.379} C_VEL
LIN {X 0,Y 320.097,Z 1143.693,A -85,B 0,C 180,E1 16419.606,E2 16419.606} C_VEL
LIN {X 0,Y 306.448,Z 1178.32,A -85,B 0,C 180,E1 16423.855,E2 16423.855} C_VEL
LIN {X 0,Y 293.889,Z 1208.033,A -85,B 0,C 180,E1 16429.104,E2 16429.104} C_VEL
LIN {X 0,Y 282.998,Z 1234.007,A -85,B 0,C 180,E1 16435.539,E2 16435.539} C_VEL
LIN {X 0,Y 275.083,Z 1255.712,A -85,B 0,C 180,E1 16443.09,E2 16443.09} C_VEL
LIN {X 0,Y 270.889,Z 1272.068,A -85,B 0,C 180,E1 16451.255,E2 16451.255} C_VEL
LIN {X 0,Y 270.001,Z 1282.264,A -85,B 0,C 180,E1 16459.092,E2 16459.092} C_VEL
LIN {X 0,Y 270.14,Z 1285.737,A -85,B 0,C 180,E1 16463.584,E2 16463.584} C_VEL
LIN {X 0,Y 270.672,Z 1287.729,A -85,B 0,C 180,E1 16469.999,E2 16469.999} C_VEL
LIN {X 0,Y 270.127,Z 1285.744,A -85,B 0,C 180,E1 16476.414,E2 16476.414} C_VEL
LIN {X 0,Y 270.029,Z 1280.128,A -85,B 0,C 180,E1 16482.915,E2 16482.915} C_VEL
LIN {X 0,Y 271.72,Z 1267.9,A -85,B 0,C 180,E1 16491.159,E2 16491.159} C_VEL
LIN {X 0,Y 277.073,Z 1249.536,A -85,B 0,C 180,E1 16499.35,E2 16499.35} C_VEL
LIN {X 0,Y 286.412,Z 1225.725,A -85,B 0,C 180,E1 16506.768,E2 16506.768} C_VEL
LIN {X 0,Y 298.418,Z 1197.626,A -85,B 0,C 180,E1 16512.954,E2 16512.954} C_VEL
LIN {X 0,Y 312.14,Z 1164.771,A -85,B 0,C 180,E1 16518.011,E2 16518.011} C_VEL
LIN {X 0,Y 325.287,Z 1129.238,A -85,B 0,C 180,E1 16521.767,E2 16521.767} C_VEL
LIN {X 0,Y 332.527,Z 1105.364,A -85,B 0,C 180,E1 16523.637,E2 16523.637} C_VEL
LIN {X 0,Y 323.598,Z 1078.979,A -85,B 0,C 180,E1 16528.804,E2 16528.804} C_VEL
LIN {X 0,Y 314.507,Z 1059.361,A -85,B 0,C 180,E1 16533.721,E2 16533.721} C_VEL
LIN {X 0,Y 309.959,Z 1054.953,A -85,B 0,C 180,E1 16535.832,E2 16535.832} C_VEL
LIN {X 0,Y 302.206,Z 1049.666,A -85,B 0,C 180,E1 16539.591,E2 16539.591} C_VEL
LIN {X 0,Y 295.636,Z 1038.892,A -85,B 0,C 180,E1 16544.576,E2 16544.576} C_VEL
LIN {X 0,Y 292.295,Z 1033.222,A -85,B 0,C 180,E1 16547.858,E2 16547.858} C_VEL
LIN {X 0,Y 288.539,Z 1026.831,A -85,B 0,C 180,E1 16552.865,E2 16552.865} C_VEL
LIN {X 0,Y 285.537,Z 1023.218,A -85,B 0,C 180,E1 16560,E2 16560} C_VEL
LIN {X 0,Y 285.25,Z 1024.485,A -85,B 0,C 180,E1 16566.073,E2 16566.073} C_VEL
LIN {X 0,Y 287.209,Z 1027.933,A -85,B 0,C 180,E1 16572.131,E2 16572.131} C_VEL
LIN {X 0,Y 290.381,Z 1035.989,A -85,B 0,C 180,E1 16578.167,E2 16578.167} C_VEL
LIN {X 0,Y 295.537,Z 1048.316,A -85,B 0,C 180,E1 16584.911,E2 16584.911} C_VEL
LIN {X 0,Y 300.972,Z 1065.342,A -85,B 0,C 180,E1 16591.762,E2 16591.762} C_VEL
LIN {X 0,Y 305.071,Z 1084.499,A -85,B 0,C 180,E1 16598.165,E2 16598.165} C_VEL
LIN {X 0,Y 306.822,Z 1103.682,A -85,B 0,C 180,E1 16603.963,E2 16603.963} C_VEL
LIN {X 0,Y 306.581,Z 1110.059,A -85,B 0,C 180,E1 16605.763,E2 16605.763} C_VEL
LIN {X 0,Y 293.084,Z 1136.662,A -85,B 0,C 180,E1 16611.49,E2 16611.49} C_VEL
LIN {X 0,Y 281.492,Z 1157.656,A -85,B 0,C 180,E1 16618.049,E2 16618.049} C_VEL
LIN {X 0,Y 272.404,Z 1173.773,A -85,B 0,C 180,E1 16625.452,E2 16625.452} C_VEL
LIN {X 0,Y 266.432,Z 1185.09,A -85,B 0,C 180,E1 16633.551,E2 16633.551} C_VEL
LIN {X 0,Y 263.945,Z 1190.562,A -85,B 0,C 180,E1 16640.125,E2 16640.125} C_VEL
LIN {X 0,Y 263.049,Z 1193.224,A -85,B 0,C 180,E1 16646.713,E2 16646.713} C_VEL
LIN {X 0,Y 263.059,Z 1193.19,A -85,B 0,C 180,E1 16653.29,E2 16653.29} C_VEL
LIN {X 0,Y 264.436,Z 1189.444,A -85,B 0,C 180,E1 16661.522,E2 16661.522} C_VEL
LIN {X 0,Y 269.058,Z 1179.96,A -85,B 0,C 180,E1 16670.521,E2 16670.521} C_VEL
LIN {X 0,Y 276.802,Z 1165.797,A -85,B 0,C 180,E1 16678.492,E2 16678.492} C_VEL
LIN {X 0,Y 287.985,Z 1145.975,A -85,B 0,C 180,E1 16685.784,E2 16685.784} C_VEL
LIN {X 0,Y 300.434,Z 1122.432,A -85,B 0,C 180,E1 16691.723,E2 16691.723} C_VEL
LIN {X 0,Y 306.779,Z 1108.567,A -85,B 0,C 180,E1 16694.521,E2 16694.521} C_VEL
LIN {X 0,Y 305.446,Z 1087.891,A -85,B 0,C 180,E1 16700.669,E2 16700.669} C_VEL
LIN {X 0,Y 302.015,Z 1069.241,A -85,B 0,C 180,E1 16706.661,E2 16706.661} C_VEL
LIN {X 0,Y 296.518,Z 1051.396,A -85,B 0,C 180,E1 16713.559,E2 16713.559} C_VEL
LIN {X 0,Y 291.507,Z 1038.412,A -85,B 0,C 180,E1 16720.06,E2 16720.06} C_VEL
LIN {X 0,Y 288.375,Z 1031.614,A -85,B 0,C 180,E1 16724.833,E2 16724.833} C_VEL
LIN {X 0,Y 286.414,Z 1026.306,A -85,B 0,C 180,E1 16729.374,E2 16729.374} C_VEL
LIN {X 0,Y 285.015,Z 1022.87,A -85,B 0,C 180,E1 16736.965,E2 16736.965} C_VEL
LIN {X 0,Y 285.895,Z 1023.903,A -85,B 0,C 180,E1 16742.269,E2 16742.269} C_VEL
LIN {X 0,Y 289.597,Z 1028.327,A -85,B 0,C 180,E1 16748.899,E2 16748.899} C_VEL
LIN {X 0,Y 293.933,Z 1035.766,A -85,B 0,C 180,E1 16753.924,E2 16753.924} C_VEL
LIN {X 0,Y 301.311,Z 1047.948,A -85,B 0,C 180,E1 16759.853,E2 16759.853} C_VEL
LIN {X 0,Y 310.719,Z 1065.819,A -85,B 0,C 180,E1 16765.917,E2 16765.917} C_VEL
LIN {X 0,Y 319.81,Z 1087.12,A -85,B 0,C 180,E1 16771.266,E2 16771.266} C_VEL
LIN {X 0,Y 326.339,Z 1109.57,A -85,B 0,C 180,E1 16775.707,E2 16775.707} C_VEL
LIN {X 0,Y 313.741,Z 1145.424,A -85,B 0,C 180,E1 16778.793,E2 16778.793} C_VEL
LIN {X 0,Y 300.399,Z 1177.795,A -85,B 0,C 180,E1 16782.864,E2 16782.864} C_VEL
LIN {X 0,Y 286.885,Z 1208.273,A -85,B 0,C 180,E1 16788.387,E2 16788.387} C_VEL
LIN {X 0,Y 275.068,Z 1235.202,A -85,B 0,C 180,E1 16795.372,E2 16795.372} C_VEL
LIN {X 0,Y 266.614,Z 1257.638,A -85,B 0,C 180,E1 16803.75,E2 16803.75} C_VEL
LIN {X 0,Y 262.763,Z 1272.863,A -85,B 0,C 180,E1 16812.12,E2 16812.12} C_VEL
LIN {X 0,Y 262.139,Z 1281.971,A -85,B 0,C 180,E1 16820.054,E2 16820.054} C_VEL
LIN {X 0,Y 262.532,Z 1285.802,A -85,B 0,C 180,E1 16826.704,E2 16826.704} C_VEL
LIN {X 0,Y 262.905,Z 1286.359,A -85,B 0,C 180,E1 16829.999,E2 16829.999} C_VEL
LIN {X 0,Y 262.31,Z 1284.356,A -85,B 0,C 180,E1 16836.606,E2 16836.606} C_VEL
LIN {X 0,Y 262.19,Z 1278.708,A -85,B 0,C 180,E1 16843.309,E2 16843.309} C_VEL
LIN {X 0,Y 263.732,Z 1267.98,A -85,B 0,C 180,E1 16850.952,E2 16850.952} C_VEL
LIN {X 0,Y 269.097,Z 1250.324,A -85,B 0,C 180,E1 16859.35,E2 16859.35} C_VEL
LIN {X 0,Y 278.535,Z 1227.107,A -85,B 0,C 180,E1 16867.018,E2 16867.018} C_VEL
LIN {X 0,Y 290.842,Z 1199.552,A -85,B 0,C 180,E1 16873.419,E2 16873.419} C_VEL
LIN {X 0,Y 304.655,Z 1168.127,A -85,B 0,C 180,E1 16878.517,E2 16878.517} C_VEL
LIN {X 0,Y 317.937,Z 1134.463,A -85,B 0,C 180,E1 16882.297,E2 16882.297} C_VEL
LIN {X 0,Y 326.417,Z 1108.232,A -85,B 0,C 180,E1 16884.485,E2 16884.485} C_VEL
LIN {X 0,Y 318.36,Z 1083.209,A -85,B 0,C 180,E1 16889.641,E2 16889.641} C_VEL
LIN {X 0,Y 307.977,Z 1060.499,A -85,B 0,C 180,E1 16895.774,E2 16895.774} C_VEL
LIN {X 0,Y 302.206,Z 1049.666,A -85,B 0,C 180,E1 16899.591,E2 16899.591} C_VEL
LIN {X 0,Y 298.148,Z 1046.781,A -85,B 0,C 180,E1 16901.916,E2 16901.916} C_VEL
LIN {X 0,Y 292.121,Z 1044.855,A -85,B 0,C 180,E1 16905.607,E2 16905.607} C_VEL
LIN {X 0,Y 291.709,Z 1044.139,A -85,B 0,C 180,E1 16906.011,E2 16906.011} C_VEL
LIN {X 0,Y 289.322,Z 1040.207,A -85,B 0,C 180,E1 16908.531,E2 16908.531} C_VEL
LIN {X 0,Y 286.086,Z 1034.275,A -85,B 0,C 180,E1 16913.184,E2 16913.184} C_VEL
LIN {X 0,Y 283.341,Z 1030.836,A -85,B 0,C 180,E1 16920,E2 16920} C_VEL
LIN {X 0,Y 282.818,Z 1032.017,A -85,B 0,C 180,E1 16926.126,E2 16926.126} C_VEL
LIN {X 0,Y 284.131,Z 1034.039,A -85,B 0,C 180,E1 16930.712,E2 16930.712} C_VEL
LIN {X 0,Y 287.393,Z 1043.72,A -85,B 0,C 180,E1 16938.362,E2 16938.362} C_VEL
LIN {X 0,Y 291.984,Z 1056.2,A -85,B 0,C 180,E1 16945.236,E2 16945.236} C_VEL
LIN {X 0,Y 296.771,Z 1074.093,A -85,B 0,C 180,E1 16952.454,E2 16952.454} C_VEL
LIN {X 0,Y 299.658,Z 1091.628,A -85,B 0,C 180,E1 16958.402,E2 16958.402} C_VEL
LIN {X 0,Y 300.569,Z 1110.261,A -85,B 0,C 180,E1 16964.216,E2 16964.216} C_VEL
LIN {X 0,Y 299.78,Z 1113.943,A -85,B 0,C 180,E1 16965.194,E2 16965.194} C_VEL
LIN {X 0,Y 286.428,Z 1139.057,A -85,B 0,C 180,E1 16970.788,E2 16970.788} C_VEL
LIN {X 0,Y 274.274,Z 1160.012,A -85,B 0,C 180,E1 16977.56,E2 16977.56} C_VEL
LIN {X 0,Y 264.379,Z 1176.677,A -85,B 0,C 180,E1 16985.647,E2 16985.647} C_VEL
LIN {X 0,Y 258.295,Z 1187.743,A -85,B 0,C 180,E1 16994.333,E2 16994.333} C_VEL
LIN {X 0,Y 255.53,Z 1193.617,A -85,B 0,C 180,E1 17003.218,E2 17003.218} C_VEL
LIN {X 0,Y 255.349,Z 1194.901,A -85,B 0,C 180,E1 17010.001,E2 17010.001} C_VEL
LIN {X 0,Y 255.525,Z 1193.565,A -85,B 0,C 180,E1 17016.784,E2 17016.784} C_VEL
LIN {X 0,Y 258.322,Z 1187.614,A -85,B 0,C 180,E1 17025.683,E2 17025.683} C_VEL
LIN {X 0,Y 264.543,Z 1176.472,A -85,B 0,C 180,E1 17034.339,E2 17034.339} C_VEL
LIN {X 0,Y 273.224,Z 1161.737,A -85,B 0,C 180,E1 17041.648,E2 17041.648} C_VEL
LIN {X 0,Y 285.09,Z 1141.415,A -85,B 0,C 180,E1 17048.458,E2 17048.458} C_VEL
LIN {X 0,Y 298.124,Z 1117.108,A -85,B 0,C 180,E1 17054.107,E2 17054.107} C_VEL
LIN {X 0,Y 300.421,Z 1111.416,A -85,B 0,C 180,E1 17055.317,E2 17055.317} C_VEL
LIN {X 0,Y 299.697,Z 1092.503,A -85,B 0,C 180,E1 17061.204,E2 17061.204} C_VEL
LIN {X 0,Y 296.667,Z 1073.499,A -85,B 0,C 180,E1 17067.588,E2 17067.588} C_VEL
LIN {X 0,Y 291.847,Z 1055.819,A -85,B 0,C 180,E1 17074.751,E2 17074.751} C_VEL
LIN {X 0,Y 286.549,Z 1041.252,A -85,B 0,C 180,E1 17082.98,E2 17082.98} C_VEL
LIN {X 0,Y 283.884,Z 1033.923,A -85,B 0,C 180,E1 17089.278,E2 17089.278} C_VEL
LIN {X 0,Y 282.759,Z 1030.48,A -85,B 0,C 180,E1 17096.941,E2 17096.941} C_VEL
LIN {X 0,Y 283.685,Z 1031.575,A -85,B 0,C 180,E1 17102.286,E2 17102.286} C_VEL
LIN {X 0,Y 287.116,Z 1035.695,A -85,B 0,C 180,E1 17108.595,E2 17108.595} C_VEL
LIN {X 0,Y 291.48,Z 1043.557,A -85,B 0,C 180,E1 17113.853,E2 17113.853} C_VEL
LIN {X 0,Y 298.61,Z 1056.143,A -85,B 0,C 180,E1 17119.944,E2 17119.944} C_VEL
LIN {X 0,Y 307.02,Z 1072.884,A -85,B 0,C 180,E1 17125.69,E2 17125.69} C_VEL
LIN {X 0,Y 315.562,Z 1094.912,A -85,B 0,C 180,E1 17131.262,E2 17131.262} C_VEL
LIN {X 0,Y 320.345,Z 1112.282,A -85,B 0,C 180,E1 17134.823,E2 17134.823} C_VEL
LIN {X 0,Y 306.315,Z 1150.053,A -85,B 0,C 180,E1 17138.265,E2 17138.265} C_VEL
LIN {X 0,Y 291.37,Z 1184.017,A -85,B 0,C 180,E1 17142.901,E2 17142.901} C_VEL
LIN {X 0,Y 277.586,Z 1213.409,A -85,B 0,C 180,E1 17148.764,E2 17148.764} C_VEL
LIN {X 0,Y 266.147,Z 1238.55,A -85,B 0,C 180,E1 17155.95,E2 17155.95} C_VEL
LIN {X 0,Y 258.375,Z 1258.469,A -85,B 0,C 180,E1 17164.064,E2 17164.064} C_VEL
LIN {X 0,Y 254.774,Z 1273.062,A -85,B 0,C 180,E1 17172.772,E2 17172.772} C_VEL
LIN {X 0,Y 254.32,Z 1280.569,A -85,B 0,C 180,E1 17179.745,E2 17179.745} C_VEL
LIN {X 0,Y 254.715,Z 1284.42,A -85,B 0,C 180,E1 17186.602,E2 17186.602} C_VEL
